// TIA Portal project "Proyecto Recreo OP 666" (V17)

(* hardware
DEVICE "S7-1200 station_1"  S7-1200 Station
   slot 0: "Rack_0"  S7-1200 Rack  Rack  V1.0
   slot 1: "PLC_1"  CPU 1214C DC/DC/DC  6ES7 214-1AG40-0XB0  V4.5
   slot 2: "DI 16/DQ 16x24VDC_1"  SM 1223 DI16/DQ16 x 24VDC  6ES7 223-1BL30-0XB0  V1.0
   slot 3: "AI 8x13BIT_1"  6ES7 231-4HF32-0XB0  V2.1
DEVICE "HMI_1"  KTP900 Basic PN
   slot 0: "HMI_1"  KTP900 Basic PN  6AV2 123-2JB03-0AX0  17.0.0.0
   slot 1: "HMI_RT_1"  KTP900 Basic PN  6AV2 123-2JB03-0AX0  17.0.0.0
   slot 5: "HMI_1.IE_CP_1"  PROFINET Interface  17.0.0.0
      slot 1: "PROFINET Interface_1"  PROFINET Interface
         slot 1: "Port_1"  Port
*)

// ===== PLC "PLC_1"  CPU 1214C DC/DC/DC =====

VAR_GLOBAL   // PLC tag table "BOOLEANAS"
   "HMI INICIAR CICLO PO" AT %M300.0 : Bool;
   "HMI INICIAR CICLO OP" AT %M300.3 : Bool;
   "HMI ON MANUAL VS" AT %M300.4 : Bool;
   "HMI ON MANUAL VV" AT %M300.5 : Bool;
   "HMI ON MANUAL CARGA AGUA" AT %M300.6 : Bool;
   "HMI ON MANUAL TOMA FILTRO" AT %M300.7 : Bool;
   "HMI ON MANUAL BALIZA VERDE" AT %M301.0 : Bool;
   "HMI ON MANUAL BALIZA ROJA" AT %M301.1 : Bool;
   "HMI ON MANUAL BUZZER" AT %M301.2 : Bool;
   "HMI SIGUIENTE EQUIPO MM" AT %M302.2 : Bool;   // Siguiente equipo modo manual
   "HMI ANTERIOR EQUIPO MM" AT %M302.3 : Bool;   // Anterior equipo modo manual
   "HMI OFF MANUAL VS" AT %M301.3 : Bool;
   "HMI OFF MANUAL VV" AT %M301.4 : Bool;
   "HMI OFF MANUAL CARGA AGUA" AT %M301.5 : Bool;
   "HMI OFF MANUAL TOMA FILTRO" AT %M301.6 : Bool;
   "HMI OFF MANUAL BALIZA VERDE" AT %M301.7 : Bool;
   "HMI OFF MANUAL BALIZA ROJA" AT %M302.0 : Bool;
   "HMI OFF MANUAL BUZZER" AT %M302.1 : Bool;
   "HMI ON MANUAL BOMBA RECIRCULACION" AT %M302.4 : Bool;
   "HMI OFF MANUAL BOMBA RECIRCULACION" AT %M302.5 : Bool;
   "HMI PAUSA" AT %M302.6 : Bool;
   "HMI CONTINUAR" AT %M302.7 : Bool;
   "HMI CANCELAR" AT %M303.0 : Bool;
   "HMI VER EQUIPO 1" AT %M303.1 : Bool;
   "HMI VER EQUIPO 2" AT %M303.2 : Bool;
   "HMI VER EQUIPO 3" AT %M303.3 : Bool;
   "HMI VER EQUIPO 4" AT %M303.4 : Bool;
   "ACTUALIZAR DATOS" AT %M303.5 : Bool;
   "HMI AUMENTAR CANT TORRES" AT %M303.6 : Bool;
   "HMI DISMINUIR CANT TORRES" AT %M303.7 : Bool;
   "HMI AUMENTAR EQUIPO" AT %M305.0 : Bool;
   "HMI DISMINUIR EQUIPO" AT %M305.1 : Bool;
   "HMI RECETA SIGUIENTE" AT %M305.2 : Bool;
   "HMI RECETA ANTERIOR" AT %M305.3 : Bool;
   "AUX 1" AT %M305.4 : Bool;
   "HMI SUMAR PASO" AT %M305.5 : Bool;
   "HMI RESTAR PASO" AT %M305.6 : Bool;
   "ACTUALIZAR RECETA" AT %M306.0 : Bool;
   "HMI SEL SIG RECETA" AT %M304.0 : Bool;
   "HMI SEL ANT RECETA" AT %M304.1 : Bool;
   "AUX 2" AT %M304.2 : Bool;
   "HMI ON BUZZER" AT %M304.3 : Bool;
   "HMI OFF BUZZER" AT %M304.4 : Bool;
   "CALIBRACION SN MAXIMO" AT %M304.5 : Bool;
   "CALIBRACION SN MINIMO" AT %M304.6 : Bool;
   "REARMADO" AT %M304.7 : Bool;
   "HMI ON LUZ PS REARME" AT %M305.7 : Bool;
   "HMI OFF LUZ PS REARME" AT %M306.1 : Bool;
   "Clock_Byte" AT %MB1500 : Byte;
   "Clock_10Hz" AT %M1500.0 : Bool;
   "Clock_5Hz" AT %M1500.1 : Bool;
   "Clock_2.5Hz" AT %M1500.2 : Bool;
   "Clock_2Hz" AT %M1500.3 : Bool;
   "Clock_1.25Hz" AT %M1500.4 : Bool;
   "Clock_1Hz" AT %M1500.5 : Bool;
   "Clock_0.625Hz" AT %M1500.6 : Bool;
   "Clock_0.5Hz" AT %M1500.7 : Bool;
   "HMI ON LUZ REARME" AT %M1501.0 : Bool;
   "HMI OFF LUZ REARME" AT %M1501.1 : Bool;
   "HMI ON INGRESO AMONIACO" AT %M306.2 : Bool;
   "HMI OFF INGRESO AMONIACO" AT %M306.3 : Bool;
   "HMI ON MANUAL V INGRESO" AT %M306.4 : Bool;
   "HMI OFF MANUAL V INGRESO" AT %M306.5 : Bool;
   "HMI ON MANUAL BI" AT %M306.6 : Bool;
   "HMI OFF MANUAL BI" AT %M306.7 : Bool;
   "HMI ON MANUAL BE" AT %M307.0 : Bool;
   "HMI OFF MANUAL BE" AT %M307.1 : Bool;
   "TIPO DE EQUIPO SELECCIONADO" AT %M307.2 : Bool;
   "HMI OK FIN DE CICLO" AT %M307.3 : Bool;
   "HMI OK CANCELAR" AT %M307.4 : Bool;
   "BLOQUEO" AT %M307.5 : Bool;
   "HMI RESET ACTUADORES MANUAL" AT %M307.6 : Bool;
   "HMI SALTAR PASO" AT %M307.7 : Bool;
   "BUZZER EQ1" AT %M308.0 : Bool;
   "BUZZER EQ2" AT %M308.1 : Bool;
   "BUZZER EQ3" AT %M308.2 : Bool;
   "BUZZER EQ4" AT %M308.3 : Bool;
   "System_Byte" AT %MB1700 : Byte;
   "FirstScan" AT %M1700.0 : Bool;
   "DiagStatusUpdate" AT %M1700.1 : Bool;
   "AlwaysTRUE" AT %M1700.2 : Bool;
   "AlwaysFALSE" AT %M1700.3 : Bool;
   "HMI VISUALIZAR RECETA" AT %M1701.0 : Bool;
   "HMI RECETARIO" AT %M1701.1 : Bool;
   "HMI VOLVER" AT %M1701.2 : Bool;
   "HMI ON LEVANTAR TAPA" AT %M1701.3 : Bool;
   "HMI OFF LEVANTAR TAPA" AT %M1701.4 : Bool;
   "HMI ON BAJAR TAPA" AT %M1701.5 : Bool;
   "HMI OFF BAJAR TAPA" AT %M1701.6 : Bool;
   "HMI CONFIRMAR LOTE" AT %M1701.7 : Bool;
END_VAR

VAR_GLOBAL   // PLC tag table "ENTERAS"
   "EQUIPO SELECCIONADO" AT %MW700 : Int;
   "EQUIPO ACTUAL" AT %MW702 : Int;
   "TORRES SELECCIONADAS" AT %MW704 : Int;
   "TORRES ACTUAL" AT %MW706 : Int;
   "CANT TORRES" AT %MW708 : Int;
   "EQUIPO MANUAL" AT %MW710 : Int;
   "AUXILIAR 1" AT %MW712 : Int;
   "AUXILIAR 2" AT %MW714 : Int;
   "AUXILIAR 3" AT %MW716 : Int;
   "AUXILIAR 4" AT %MW718 : Int;
   "AUXILIAR 5" AT %MW720 : Int;
   "TEMP CORTE PC" AT %MW726 : Int;
   "TIEMPO CORTE PC" AT %MW728 : Int;
   "CORTE PC POR TEMP" AT %MW730 : Int;
   "CORTE PC POR TIEMPO" AT %MW732 : Int;
   "DELAY" AT %MW734 : Int;
   "NM_CT" AT %MW736 : Int;   // Nivel minimo segun cantidad de torres
   "CTD PASADAS" AT %MW738 : Int;   // Cantidad de pasadas
   "FLAG CR" AT %MW740 : Int;   // Flag calculos realizados
   "HMI NUMERO RECETA" AT %MW742 : Int;
   "EQUIPO ACTUAL CALCULO" AT %MW744 : Int;
   "HMI RECETA SELECCIONADA" AT %MW746 : Int;
   "HMI NIVEL" AT %MW748 : Int;
   "AUXILIAR 6" AT %MW750 : Int;
   "VER NUMERO RECETA" AT %MW752 : Int;
   "VALOR CONTRASEÑA CALCULADA" AT %MD754 : DInt;
   "HMI CONTRASEÑA INGRESADA" AT %MD758 : DInt;
   "DIAS RESTANTES" AT %MD762 : DInt;
   "DIAS TRANSCURRIDOS" AT %MD766 : DInt;
   "IMAGEN BLOQUEO" AT %MW770 : Int;
   "AUX REC SEL" AT %MW772 : Int;
   "AUX NUM REC" AT %MW774 : Int;
END_VAR

VAR_GLOBAL   // PLC tag table "Entradas Analogicas"
   "PT100 agua EQ1" AT %IW96 : Int;
   "PT100 ingreso EQ1" AT %IW98 : Int;
   "PT100 producto EQ1" AT %IW100 : Int;
   "Regla nivel EQ1" AT %IW64 : Int;
   "PT100 agua EQ2" AT %IW104 : Int;
   "PT100 ingreso EQ2" AT %IW106 : Int;
   "PT100 producto EQ2" AT %IW108 : Int;
   "Regla nivel EQ2" AT %IW66 : Int;
END_VAR

VAR_GLOBAL   // PLC tag table "Salidas digitales"
   "C1 VS" AT %Q20.3 : Bool;
   "C1 VV" AT %Q20.4 : Bool;
   "C1 CARGA DE AGUA" AT %Q20.1 : Bool;
   "C1 BOMBA" AT %Q20.0 : Bool;
   "C1 BALIZA ROJA" AT %Q0.0 : Bool;
   "C1 BALIZA VERDE" AT %Q0.1 : Bool;
   "BUZZER" AT %Q0.4 : Bool;
   "C1 TOMA FILTRO" AT %Q20.2 : Bool;
   "LUZ PS REARME" AT %Q0.5 : Bool;
   "E1 BALIZA ROJA" AT %Q0.2 : Bool;
   "E1 BALIZA VERDE" AT %Q0.3 : Bool;
   "E1 CARGA DE AGUA" AT %Q20.6 : Bool;
   "E1 TOMA FILTRO" AT %Q20.7 : Bool;
   "E1 BOMBA" AT %Q20.5 : Bool;
   "E1 INGRESO AMONIACO" AT %Q21.0 : Bool;
   "LEVANTAR TAPA" AT %Q21.1 : Bool;   // VER DIRECCION
   "CERRAR TAPA" AT %Q0.6 : Bool;   // VER DIRECCION
END_VAR

VAR_GLOBAL   // PLC tag table "Entradas digitales"
   "VVC_C" AT %I0.2 : Bool;   // True en Reposo
   "VVA_C" AT %I0.3 : Bool;   // True cuando esta activada
   "VSC_C" AT %I0.6 : Bool;   // True en reposo
   "VSA_C" AT %I0.7 : Bool;   // True cuando esta activada
   "ESTADO REARME" AT %I6.0 : Bool;   // Estado de rearme ( Circuito si o no rearmado)
   "PRARM" AT %I1.0 : Bool;   // Pulsador de rearme
   "PEMERG" AT %I1.2 : Bool;   // Pulsador parada de emergencia
   "CH_F_E" AT %I1.3 : Bool;   // Falla chiller enfriador
   "GM_E" AT %I20.0 : Bool;   // Guardamotor bomba enfriador
   "GM_C" AT %I20.1 : Bool;   // Guardamotor bomba cocina
   "PS SUBIR TAPA" AT %I20.2 : Bool;
   "PS BAJAR TAPA" AT %I20.3 : Bool;
END_VAR

DATA_BLOCK "FUNCION EQUIPO_DB"   // DB2
{ S7_Optimized_Access := 'TRUE' }
VERSION : 0.1
// stored: InstanceOfName FUNCION EQUIPO
"FUNCION EQUIPO"
BEGIN
END_DATA_BLOCK

DATA_BLOCK "NOMBRE DE LOS EQUIPOS"   // DB3
{ S7_Optimized_Access := 'TRUE' }
VERSION : 0.1
   VAR
      EQUIPOS : Array[1..2] of String;
   END_VAR
BEGIN
   EQUIPOS[1] := 'COCINA 1';
   EQUIPOS[2] := 'ENFRIADOR 1';
END_DATA_BLOCK

DATA_BLOCK "ESTRUCTURAS Y ARREGLOS"   // DB4
{ S7_Optimized_Access := 'TRUE' }
VERSION : 0.1
   VAR
      TEMPERATURAS : Array[1..2] of Struct
         "TEMPERATURA AGUA" : Real;
         "TEMPERATURA INGRESO" : Real;
         "TEMPERATURA PRODUCTO" : Real;
         "TEMPERATURA AGUA SC" : Real;
         "TEMPERATURA INGRESO SC" : Real;
         "TEMPERATURA PRODUCTO SC" : Real;
      END_STRUCT;
      NIVEL : Array[1..2] of Int;
   END_VAR
   VAR RETAIN
      CORRECCIONES : Array[1..2] of Struct
         "TEMPERATURA AGUA" : Real;
         "TEMPERATURA INGRESO" : Real;
         "TEMPERATURA PRODUCTO" : Real;
      END_STRUCT;
   END_VAR
   VAR
      "NIVEL ALCANZADO" : Array[1..2] of Bool;
   END_VAR
   VAR RETAIN
      "TEMP CORTE PO" : Array[1..4] of Int;
      CONFIGURACION : Array[1..2] of Struct
         DELAY : Int;
         HISTERESIS : DInt;
         "TIEMPO MAXIMO CICLO" : Int;
         "NIVEL CRITICO PO" : Int;
         "NIVEL PO" : Array[1..3] of Int;
         "NIVEL OP" : Int;
         VENTANA : Int;
         "NIVEL CRITICO OP" : Int;
      END_STRUCT;
   END_VAR
   VAR
      "HMI CONFIGURACION" : Struct
         DELAY : Int;
         HISTERESIS : DInt;
         "TIEMPO MAXIMO CICLO" : Int;
         "NIVEL CRITICO PO" : Int;
         "NIVEL PO" : Array[1..3] of Int;
         "NIVEL OP" : Int;
         VENTANA : Int;
         "NIVEL CRITICO OP" : Int;
      END_STRUCT;
   END_VAR
   VAR RETAIN
      CARGA : Array[1..2] of Struct   // Lo traslado a cada equipo desde HMI carga
         "CANTIDAD DE TORRES" : Int;
         "NIVEL MINIMO" : Array[1..3] of Int;   // El arreglo es porque hay 3 torres
         "TIPO DE CORTE" : Bool;
         "TEMPERATURA CORTE PC" : Int;
         "TIEMPO CORTE PC" : Int;
         "NUMERO RECETA" : Int;
         "NOMBRE RECETA" : String;
         "ESTADO ACTUAL" : String;
         "TIEMPO TOTAL TRANSCURRIDO" : Int;
         "PASO ACTUAL" : Int;
         "VAPOR VIVO" : Bool;
      END_STRUCT;
   END_VAR
   VAR
      "HMI CARGA" : Struct   // Lo que veo en la pantalla cuando selecciono cada equipo (comun a todos)
         TEMPERATURAS : Struct
            "TEMPERATURA AGUA" : Real;
            "TEMPERATURA INGRESO" : Real;
            "TEMPERATURA PRODUCTO" : Real;
            "TEMPERATURA AGUA SC" : Real;
            "TEMPERATURA INGRESO SC" : Real;
            "TEMPERATURA PRODUCTO SC" : Real;
         END_STRUCT;
         NIVEL : Int;
         "CANTIDAD DE TORRES" : Int := 1;
         "NIVEL MINIMO" : Int;
         "TIPO DE CORTE" : Bool;
         "TEMPERATURA CORTE PC" : Int;
         "TIEMPO CORTE PC" : Int;
         "NUMERO RECETA" : Int;
         "NOMBRE RECETA" : String;
         "ESTADO ACTUAL" : String;
         "TIEMPO TOTAL TRANSCURRIDO" : Int;
         "PASO ACTUAL" : Int;
         "VAPOR VIVO" : Bool;
      END_STRUCT;
      "HMI EDICION RECETAS" : Struct
         PASOS : Int;
         "TEMP AGUA" : Array[1..4] of Int;
         "TEMP PRODUCTO" : Array[1..4] of Int;
         "TIEMPO CORTE" : Array[1..4] of Int;
         "TIPO CORTE" : Array[1..4] of Bool;
         NOMBRE : String;
         "TIEMPO CORTE ENFRIADO" : Int;
         "TEMP CORTE ENFRIADO" : Int;
         "TIPO CORTE ENFRIADO" : Bool;
      END_STRUCT;
   END_VAR
   VAR RETAIN
      RECETARIO : Array[0..20] of Struct
         PASOS : Int;
         "TEMP AGUA" : Array[1..4] of Int;
         "TEMP PRODUCTO" : Array[1..4] of Int;
         "TIEMPO CORTE" : Array[1..4] of Int;
         "TIPO CORTE" : Array[1..4] of Bool;
         NOMBRE : String;
         "TIEMPO CORTE ENFRIADO" : Int;
         "TEMP CORTE ENFRIADO" : Int;
         "TIPO CORTE ENFRIADO" : Bool;
      END_STRUCT;
      "CARGA RECETA" : Array[1..2] of Struct   // Se guarda la receta elegida en cada equipo
         PASOS : Int;
         "TEMP AGUA" : Array[1..4] of Int;
         "TEMP PRODUCTO" : Array[1..4] of Int;
         "TIEMPO CORTE" : Array[1..4] of Int;
         "TIPO CORTE" : Array[1..4] of Bool;
         NOMBRE : String;
         "TIEMPO CORTE ENFRIADO" : Int;
         "TEMP CORTE ENFRIADO" : Int;
         "TIPO CORTE ENFRIADO" : Bool;
      END_STRUCT;
      "CARGA NUMERO RECETA" : Array[0..4] of Int;   // *********** CUIDADOOOO
   END_VAR
   VAR
      "CORRECCIONES HMI" : Struct
         "TEMPERATURA AGUA SC" : Real;
         "TEMPERATURA INGRESO SC" : Real;
         "TEMPERATURA PRODUCTO SC" : Real;
      END_STRUCT;
      "CALIBRAR MINIMO SN" : Array[1..2] of Bool;
      "CALIBRAR MAXIMO SN" : Array[1..2] of Bool;
      "HMI MOSTRAR RECETA" : Struct
         PASOS : Int;
         "TEMP AGUA" : Array[1..4] of Int;
         "TEMP PRODUCTO" : Array[1..4] of Int;
         "TIEMPO CORTE" : Array[1..4] of Int;
         "TIPO CORTE" : Array[1..4] of Bool;
         NOMBRE : String;
         "TIEMPO CORTE ENFRIADO" : Int;
         "TEMP CORTE ENFRIADO" : Int;
         "TIPO CORTE ENFRIADO" : Int;
      END_STRUCT;
      "HMI ESTADO" : Struct
         EQUIPO : String;
         CHILLER : String;
         "COLOR EN HMI" : Int;
         "TIEMPO TRANSCURRIDO" : DInt;
         "EN PO" : Bool;
         "EN OP" : Bool;
         "EN CICLO" : Bool;
         "TIPO DE CORTE" : String;
         "PULSADOR PAUSA" : Bool;
         "PULSADOR CONTINUAR" : Bool;
         "PULSADOR CANCELAR" : Bool;
         "CICLO CANCELADO" : Bool;
         "CICLO FINALIZADO" : Bool;
         "PULSADOR CICLO CANCELADO" : Bool;
         "PULSADOR CICLO FINALIZADO" : Bool;
         "RESET ACTUADORES" : Bool;
         "MANUAL ACTIVO" : Bool;
         "PASO ACTUAL" : Int;
      END_STRUCT;
      ESTADO : Array[1..2] of Struct
         EQUIPO : String;
         CHILLER : String;
         "COLOR EN HMI" : Int;
         "TIEMPO TRANSCURRIDO" : DInt;
         "EN PO" : Bool;
         "EN OP" : Bool;
         "EN CICLO" : Bool;
         "TIPO DE CORTE" : String;
         "PULSADOR PAUSA" : Bool;
         "PULSADOR CONTINUAR" : Bool;
         "PULSADOR CANCELAR" : Bool;
         "CICLO CANCELADO" : Bool;
         "CICLO FINALIZADO" : Bool;
         "PULSADOR CICLO CANCELADO" : Bool;
         "PULSADOR CICLO FINALIZADO" : Bool;
         "RESET ACTUADORES" : Bool;
         "MANUAL ACTIVO" : Bool;
         "PASO ACTUAL" : Int;
         "CONFIRMACION LOTE" : Bool;
      END_STRUCT;
      "HMI NOMBRE EQUIPO" : String;
   END_VAR
BEGIN
   CARGA[1]."CANTIDAD DE TORRES" := 1;
   CARGA[2]."CANTIDAD DE TORRES" := 1;
   CONFIGURACION[1]."NIVEL PO"[1] := 1020;   // Nivel PO para 1 torre
   CONFIGURACION[1]."NIVEL PO"[2] := 825;   // Nivel PO para 2 torres
   CONFIGURACION[1]."NIVEL PO"[3] := 700;   // Nivel PO para 3 torres
   CONFIGURACION[1].HISTERESIS := 2;
   CONFIGURACION[1]."TIEMPO MAXIMO CICLO" := 400;
   CONFIGURACION[2].HISTERESIS := 2;
   CONFIGURACION[2]."TIEMPO MAXIMO CICLO" := 400;
   CONFIGURACION[2]."NIVEL PO"[1] := 1020;
   CONFIGURACION[2]."NIVEL PO"[2] := 825;
   CONFIGURACION[2]."NIVEL PO"[3] := 700;
   CONFIGURACION[1]."NIVEL OP" := 1163;
   CONFIGURACION[2]."NIVEL OP" := 1163;
   CONFIGURACION[2]."NIVEL CRITICO PO" := 550;
   CONFIGURACION[2]."NIVEL CRITICO OP" := 985;
   // "HMI CONFIGURACION"."NIVEL PO"[1] : Nivel para 1 torre
   // "HMI CONFIGURACION"."NIVEL PO"[2] : Nivel para 2 torres
   // "HMI CONFIGURACION"."NIVEL PO"[3] : Nivel para 3 torres
   // CARGA[1] : Cada equipo con sus configuraciones en
END_DATA_BLOCK

DATA_BLOCK "ALARMAS"   // DB5
{ S7_Optimized_Access := 'FALSE' }
VERSION : 0.1
   VAR
      COCINAS : Struct
         "FALLA VALVULA VAPOR SERPENTINA" : Bool;
         "FALLA VALVULA VAPOR VIVO" : Bool;
         "FALLA GUARDAMOTOR" : Bool;
         "NIVEL CRITICO" : Bool;
         "FALLA SENSOR TEMP AGUA" : Bool;
         "FALLA SENSOR TEMP INGRESO" : Bool;
         "FALLA SENSOR TEMP PRODUCTO" : Bool;
         "TIEMPO MAXIMO CARGA DE AGUA" : Bool;
      END_STRUCT;
      ENFRIADOR : Struct
         "FALLA GUARDAMOTOR" : Bool;
         "FALLA CHILLER" : Bool;
         "NIVEL CRITICO" : Bool;
         "FALLA SENSOR TEMP AGUA" : Bool;
         "FALLA SENSOR TEMP INGRESO" : Bool;
         "FALLA SENSOR TEMP PRODUCTO" : Bool;
         "TIEMPO MAXIMO CARGA DE AGUA" : Bool;
      END_STRUCT;
      "PULSADOR EM ACTIVO" : Bool;
      "PRESIONAR PULSADOR REARME" : Bool;
   END_VAR
BEGIN
END_DATA_BLOCK

DATA_BLOCK "ENTRADAS Y SALIDAS"   // DB6
{ S7_Optimized_Access := 'TRUE' }
VERSION : 0.1
   VAR
      "VV MANUAL" : Array[1..2] of Bool;
      "VS MANUAL" : Array[1..2] of Bool;
      "CARGA AGUA MANUAL" : Array[1..2] of Bool;
      "TOMA FILTRO MANUAL" : Array[1..2] of Bool;
      "BOMBA RECIRCULACION MANUAL" : Array[1..2] of Bool;
      "BALIZA VERDE MANUAL" : Array[1..2] of Bool;
      "BALIZA ROJA MANUAL" : Array[1..2] of Bool;
      "INGRESO AMONIACO MANUAL" : Array[1..2] of Bool;
      "LEVANTAR TAPA MANUAL" : Array[1..2] of Bool;
      "BAJAR TAPA MANUAL" : Array[1..2] of Bool;
      "INGRESO AMONIACO" : Array[1..2] of Bool;
      GUARDAMOTOR : Array[1..2] of Bool;
      "SERPENTINA ABIERTA" : Array[1..2] of Bool;
      "SERPENTINA CERRADA" : Array[1..2] of Bool;
      "VAPOR VIVO ABIERTO" : Array[1..2] of Bool;
      "VAPOR VIVO CERRADO" : Array[1..2] of Bool;
      "FALLA CHILLER" : Array[1..2] of Bool;
      "BUZZER MANUAL" : Bool;
      "LUZ MANUAL PS REARME" : Bool;
   END_VAR
BEGIN
END_DATA_BLOCK

DATA_BLOCK "ESTADO"   // DB7
{ S7_Optimized_Access := 'TRUE' }
VERSION : 0.1
   VAR
      SALIDAS : Struct
         COCINAS : Array[1..2] of Struct
            "BALIZA VERDE" : Bool;
            "BALIZA ROJA" : Bool;
            "BOMBA RECIRCULACION" : Bool;
            "CARGA DE GUA" : Bool;
            "TOMA FILTRO" : Bool;
            "VAPOR SERPENTINA" : Bool;
            "VAPOR VIVO" : Bool;
         END_STRUCT;
         ENFRIADORES : Array[1..2] of Struct
            "BALIZA VERDE" : Bool;
            "BALIZA ROJA" : Bool;
            "BOMBA RECIRCULACION" : Bool;
            "CARGA DE AGUA" : Bool;
            "TOMA FILTRO" : Bool;
            "INGRESO AMONIACO" : Bool;
         END_STRUCT;
      END_STRUCT;
      ENTRADAS : Struct
         COCINAS : Array[1..2] of Struct
            GUARDAMOTOR : Bool;
            "VAPOR VIVO CERRADO" : Bool;
            "VAPOR VIVO ABIERTO" : Bool;
            "SERPENTINA CERRADA" : Bool;
            "SERPENTINA ABIERTA" : Bool;
         END_STRUCT;
         ENFRIADORES : Array[1..2] of Struct
            GUARDAMOTOR : Bool;
            "FALLA CHILLER" : Bool;
         END_STRUCT;
      END_STRUCT;
   END_VAR
BEGIN
END_DATA_BLOCK

DATA_BLOCK "VISUALIZACIONES HMI"   // DB8
{ S7_Optimized_Access := 'TRUE' }
VERSION : 0.1
   VAR
      "ON VS" : Bool;
      "OFF VS" : Bool;
      "ON VV" : Bool;
      "OFF VV" : Bool;
      "ON/OFF CARGA AGUA" : Bool;
      "ON/OFF TOMA FILTRO" : Bool;
      "ON/OFF BOMBA RECIRCULACION" : Bool;
      "ON/OFF BV" : Bool;
      "ON/OFF BR" : Bool;
      "ON BOMBA INGRESO" : Bool;
      "OFF BOMBA INGRESO" : Bool;
      "ON BOMBA EGRESO" : Bool;
      "OFF BOMBA EGRESO" : Bool;
      "ON V INGRESO" : Bool;
      "OFF V INGRESO" : Bool;
      "ON V EGRESO" : Bool;
      "OFF V EGRESO" : Bool;
      "ON SUBIR TAPA" : Bool;
      "OFF SUBIR TAPA" : Bool;
      "ON BAJAR TAPA" : Bool;
      "OFF BAJAR TAPA" : Bool;
      "ON INGRESO AMONIACO" : Bool;
      "OFF INGRESO AMONIACO" : Bool;
      BUZZER : Bool;
      "GUARDAMOTOR BOMBA REC" : Bool;
      "SERPENTINA CERRADA" : Bool;
      "SERPENTINA ABIERTA" : Bool;
      "VAPOR VIVO CERRADO" : Bool;
      "VAPOR VIVO ABIERTO" : Bool;
      "NV CHILLER REBALSE" : Bool;
      "NV CHILLER OK" : Bool;
      "NV CHILLER BAJO" : Bool;
      "GUARDAMOTOR BOMBA INGRESO" : Bool;
      "GUARDAMOTOR BOMBA EGRESO" : Bool;
      "FALLA CHILLER" : Bool;
      "1 PASO RECETA" : Bool;
      "2 PASOS RECETA" : Bool;
      "3 PASOS RECETA" : Bool;
      "4 PASOS RECETA" : Bool;
      "CORTE TEMP PASO 1" : Bool;
      "CORTE TEMP PASO 2" : Bool;
      "CORTE TEMP PASO 3" : Bool;
      "CORTE TEMP PASO 4" : Bool;
      "CORTE TIEMPO PASO 1" : Bool;
      "CORTE TIEMPO PASO 2" : Bool;
      "CORTE TIEMPO PASO 3" : Bool;
      "CORTE TIEMPO PASO 4" : Bool;
      "CORTE TEMP ENFRIADOR" : Bool;
      "CORTE TIEMPO ENFRIADOR" : Bool;
      "PASOS OP EN COCINAS" : Bool;
      GRAFICOS : Int;
      "LIM SUP CANT TORRES" : Bool;
      "LIM INF CANT TORRES" : Bool;
      "LIM SUP EQUIPO SEL" : Bool;
      "LIM INF EQUIPO SEL" : Bool;
      "EN VISUALIZAR RECETA" : Bool;
      "EN RECETARIO" : Bool;
      "SIGUIENTE RECETA" : Bool;
      "ANTERIOR RECETA" : Bool;
      "SIGUIENTE PASO" : Bool;
      "ANTERIOR PASO" : Bool;
      "BLOQUEO EDICION RECETAS" : Bool;
   END_VAR
BEGIN
END_DATA_BLOCK

DATA_BLOCK "SELECCION DE EQUIPO_DB"   // DB9
{ S7_Optimized_Access := 'TRUE' }
VERSION : 0.1
// stored: InstanceOfName SELECCION DE EQUIPO
"SELECCION DE EQUIPO"
BEGIN
END_DATA_BLOCK

DATA_BLOCK "EQUIPO 1"   // DB10
{ S7_Optimized_Access := 'TRUE' }
VERSION : 0.1
// stored: InstanceOfName NIVEL DE AGUA
"NIVEL DE AGUA"
BEGIN
END_DATA_BLOCK

DATA_BLOCK "EQUIPO 2"   // DB14
{ S7_Optimized_Access := 'TRUE' }
VERSION : 0.1
// stored: InstanceOfName NIVEL DE AGUA
"NIVEL DE AGUA"
BEGIN
END_DATA_BLOCK

DATA_BLOCK "EQUIPO 3"   // DB15
{ S7_Optimized_Access := 'TRUE' }
VERSION : 0.1
// stored: InstanceOfName NIVEL DE AGUA
"NIVEL DE AGUA"
BEGIN
END_DATA_BLOCK

DATA_BLOCK "EQUIPO 4"   // DB16
{ S7_Optimized_Access := 'TRUE' }
VERSION : 0.1
// stored: InstanceOfName NIVEL DE AGUA
"NIVEL DE AGUA"
BEGIN
END_DATA_BLOCK

DATA_BLOCK "EQUIPO_3"   // DB17
{ S7_Optimized_Access := 'TRUE' }
VERSION : 0.1
// stored: InstanceOfName ENFRIADOR
"ENFRIADOR"
BEGIN
END_DATA_BLOCK

DATA_BLOCK "SENSADO ENTRADA FUNCION"   // DB18
{ S7_Optimized_Access := 'TRUE' }
VERSION : 0.1
   VAR
      ENFRIADORES : Struct
         "GUARDAMOTOR BI" : Array[1..4] of Bool;
         "GUARDAMOTOR BE" : Array[1..4] of Bool;
         "NIVEL BAJO CHILLER" : Array[1..4] of Bool;
         "NIVEL OK CHILLER" : Array[1..4] of Bool;
         "NIVEL REBALSE CHILLER" : Array[1..4] of Bool;
         "FALLA CHILLER" : Array[1..4] of Bool;
      END_STRUCT;
   END_VAR
BEGIN
END_DATA_BLOCK

DATA_BLOCK "EQUIPO_4"   // DB19
{ S7_Optimized_Access := 'TRUE' }
VERSION : 0.1
// stored: InstanceOfName ENFRIADOR
"ENFRIADOR"
BEGIN
END_DATA_BLOCK

DATA_BLOCK "EQUIPO_1"   // DB20
{ S7_Optimized_Access := 'TRUE' }
VERSION : 0.1
// stored: InstanceOfName COCINA
"COCINA"
BEGIN
END_DATA_BLOCK

DATA_BLOCK "EQUIPO_2"   // DB21
{ S7_Optimized_Access := 'TRUE' }
VERSION : 0.1
// stored: InstanceOfName COCINA
"COCINA"
BEGIN
END_DATA_BLOCK

DATA_BLOCK "Coordinacion"   // DB22
{ S7_Optimized_Access := 'TRUE' }
VERSION : 0.1
   VAR
      Comunicacion : Int;
   END_VAR
BEGIN
END_DATA_BLOCK

DATA_BLOCK "COMUNICACION"   // DB23
{ S7_Optimized_Access := 'TRUE' }
VERSION : 0.1
   VAR
      ESTADO : Int;
      "T AGUA" : Real;
      "T INGRESO" : Real;
      "T PROD" : Real;
      NIVEL : Int;
      "NOMBRE RECETA" : String;
      "NUMERO RECETA" : Int;
      "NUMERO EQUIPO" : Int;
      SERPENTINA : Bool;
      "VAPOR VIVO" : Bool;
      TORRES : Int;
      PASOS : Int;
      "TIEMPO TRANSCURRIDO" : DInt;
   END_VAR
BEGIN
END_DATA_BLOCK

DATA_BLOCK "ENVIO EQUIPO 1"   // DB24
{ S7_Optimized_Access := 'TRUE' }
VERSION : 0.1
// stored: InstanceOfName ENVIO DATOS
"ENVIO DATOS"
BEGIN
END_DATA_BLOCK

// folder: System blocks/Program resources

DATA_BLOCK "CANTIDAD TORRES"   // DB1
{ S7_Optimized_Access := 'TRUE' }
AUTHOR : Simatic
FAMILY : IEC
NAME : CNTR
VERSION : 1.0
// stored: InstanceOfName IEC_COUNTER
"IEC_COUNTER"
BEGIN
END_DATA_BLOCK

DATA_BLOCK "CONTADOR RECETAS"   // DB11
{ S7_Optimized_Access := 'TRUE' }
AUTHOR : Simatic
FAMILY : IEC
NAME : CNTR
VERSION : 1.0
// stored: InstanceOfName IEC_COUNTER
"IEC_COUNTER"
BEGIN
END_DATA_BLOCK

DATA_BLOCK "CONTADOR PASOS"   // DB12
{ S7_Optimized_Access := 'TRUE' }
AUTHOR : Simatic
FAMILY : IEC
NAME : CNTR
VERSION : 1.0
// stored: InstanceOfName IEC_COUNTER
"IEC_COUNTER"
BEGIN
END_DATA_BLOCK

DATA_BLOCK "CONTADOR SELECCION DE RECETA"   // DB13
{ S7_Optimized_Access := 'TRUE' }
AUTHOR : Simatic
FAMILY : IEC
NAME : CNTR
VERSION : 1.0
// stored: InstanceOfName IEC_COUNTER
"IEC_COUNTER"
BEGIN
END_DATA_BLOCK

// folder: (top level)

FUNCTION_BLOCK "ENFRIADOR"   // FB1, LAD
{ S7_Optimized_Access := 'TRUE' }
VERSION : 0.1
   VAR_INPUT
      REARME : Bool;
      "PARAMETROS CICLOS" : Struct
         "CANTIDAD DE TORRES" : Int;
         "NIVEL MINIMO" : Array[1..3] of Int;   // El arreglo es porque hay 3 torres
         "TIPO DE CORTE" : Bool;
         "TEMPERATURA CORTE PO" : Int;
         "TIEMPO CORTE PO" : Int;
         "NUMERO RECETA" : Int;
         "NOMBRE RECETA" : String;
         "ESTADO ACTUAL" : String;
         "TIEMPO TOTAL TRANSCURRIDO" : Int;
         "PASO ACTUAL" : Int;
         "VAPOR VIVO" : Bool;
      END_STRUCT;
      CONFIGURACION : Struct
         DELAY : Int;
         HISTERESIS : DInt;
         "TIEMPO MAXIMO CICLO" : Int;
         "NIVEL CRITICO" : Int;
         "NIVEL PO" : Array[1..3] of Int;
         "NIVEL OP" : Int;
         VENTANA : Int;
         "NIVEL CRITICO OP" : Int;
      END_STRUCT;
      RECETA : Struct
         PASOS : Int;
         "TEMP AGUA" : Array[1..4] of Int;
         "TEMP PRODUCTO" : Array[1..4] of Int;
         "TIEMPO CORTE" : Array[1..4] of Int;
         "TIPO CORTE" : Array[1..4] of Bool;
         NOMBRE : String;
         "TIEMPO CORTE ENFRIADO" : Int;
         "TEMP CORTE ENFRIADO" : Int;
         "TIPO CORTE ENFRIADO" : Bool;
      END_STRUCT;
      TEMPERATURAS : Struct
         "TEMPERATURA AGUA" : Real;
         "TEMPERATURA INGRESO" : Real;
         "TEMPERATURA PRODUCTO" : Real;
         "TEMPERATURA AGUA SC" : Real;
         "TEMPERATURA INGRESO SC" : Real;
         "TEMPERATURA PRODUCTO SC" : Real;
      END_STRUCT;
      NIVEL : Int;
      GUARDAMOTOR : Bool;
      "MANUAL BALIZA VERDE" : Bool;
      "MANUAL BALIZA ROJA" : Bool;
      "MANUAL BOMBA" : Bool;
      "MANUAL CARGA DE AGUA" : Bool;
      "MANUAL TOMA FILTRO" : Bool;
      "MANUAL INGRESO AMONIACO" : Bool;
      "EQUIPO SELECCIONADO" : Int;
      "NUMERO DE EQUIPO" : Int;
      "INICIAR PRE OPERATIVO" : Bool;
      "INICIAR OPERATIVO" : Bool;
      PAUSA : Bool;
      CONTINUAR : Bool;
      CANCELAR : Bool;
      "PULSADOR EMERGENCIA" : Bool;
      "OK FIN CICLO" : Bool;
      "OK CANCELAR" : Bool;
      "RESET ACTUADORES EN MANUAL" : Bool;
   END_VAR
   VAR_OUTPUT
      "BALIZA VERDE" : Bool;
      "BALIZA ROJA" : Bool;
      BUZER : Bool;
      BOMBA : Bool;
      "CARGA DE AGUA" : Bool;
      "TOMA FILTRO" : Bool;
      "INGRESO AMONIACO" : Bool;
      ESTADO : Struct
         EQUIPO : String;
         CHILLER : String;
         "COLOR EN HMI" : Int;
         "TIEMPO TRANSCURRIDO" : DInt;
         "EN PO" : Bool;
         "EN OP" : Bool;
         "EN CICLO" : Bool;
         "TIPO DE CORTE" : String;
         "PULSADOR PAUSA" : Bool;
         "PULSADOR CONTINUAR" : Bool;
         "PULSADOR CANCELAR" : Bool;
         "CICLO CANCELADO" : Bool;
         "CICLO FINALIZADO" : Bool;
         "PULSADOR CICLO CANCELADO" : Bool;
         "PULSADOR CICLO FINALIZADO" : Bool;
         "RESET ACTUADORES" : Bool;
         "MANUAL ACTIVO" : Bool;
         "PASO ACTUAL" : Int;
      END_STRUCT;
      ALARMAS : Struct
         "FALLA GUARDAMOTOR" : Bool;
         "FALLA CHILLER" : Bool;
         "NIVEL CRITICO TANQUE" : Bool;
         "FALLA SENSOR TEMP AGUA" : Bool;
         "FALLA SENSOR TEMP INGRESO" : Bool;
         "FALLA SENSOR TEMP PRODUCTO" : Bool;
         "TIEMPO MAXIMO CARGA DE AGUA" : Bool;
      END_STRUCT;
      "ESTADO ENTRADAS" : Struct
         GUARDAMOTOR : Bool;
         "FALLA CHILLER" : Bool;
      END_STRUCT;
      "ESTADO SALIDAS" : Struct
         "BALIZA VERDE" : Bool;
         "BALIZA ROJA" : Bool;
         "BOMBA RECIRCULACION" : Bool;
         "CARGA DE AGUA" : Bool;
         "TOMA FILTRO" : Bool;
         "INGRESO AMONIACO" : Bool;
      END_STRUCT;
   END_VAR
   VAR
      HABILITADO : Bool;
      "EN FALLA" : Bool;
      "CICLO PO ACTIVO" : Bool;
      "CICLO CANCELADO" : Bool;
      "CICLO PAUSADO" : Bool;
      "NIVEL PO" : Int;
      "TEMPERATURA PO ALCANZADA" : Bool;
      "TIEMPO PO" : TON_TIME;
      "TIEMPO CORTE PO" : DInt;
      "TIEMPO PO ALCANZADO" : Bool;
      "FIN CICLO PO" : Bool;
      "CICLO OP ACTIVO" : Bool;
      "TEMPERATURA OP ALCANZADA" : Bool;
      "TIEMPO OP" : TONR_TIME;
      "TIEMPO CORTE OP" : DInt;
      "FALTA AGUA PARA CHILLER" : Bool;
      "NIVEL CH CORRECTO COMIENZO" : Bool;
      "V EGRESO PARA CARGA CH" : Bool;
      "MANDAR AGUA A CH" : Bool;
      "CARGAR AGUA TQ PARA CARGA CH" : Bool;
      "CARGA AGUA TQ" : Bool;
      "NIVEL TQ ALCANZADO" : Bool;
      "NIVEL MINIMO" : Int;
      "NIVEL MAXIMO" : Int;
      "EN RANGO" : Bool;
      "NIVEL DEBAJO MINIMO" : Bool;
      "NIVEL SUPERA MAXIMO" : Bool;
      BOMBA_EGRESO : TON_TIME;
      BOMBA_INGRESO : TON_TIME;
      IEC_Timer_0_Instance : TOF_TIME;
      IEC_Timer_0_Instance_1 : TOF_TIME;
      DELAYS : DInt;
      "EN NIVEL PARA BI" : Bool;
      "EN NIVEL PARA BE" : Bool;
      "NIVEL TRABAJO" : Int;
      "NIVEL PARA CARGA DE AGUA" : Int;
      "TIEMPO OP ALCANZADO" : Bool;
      "FIN CICLO OP" : Bool;
      F1 : Bool;
      F2 : Bool;
      "TIEMPO MAXIMO" : DInt;
      AUXILIAR : DInt;
      IEC_Timer_0_Instance_2 : TONR_TIME;
      "CICLO PO FINALIZADO" : Bool;
      "CICLO OP FINALIZADO" : Bool;
      "ACTUADORES MANUALES ACTIVOS" : Bool;
      IEC_Timer_0_Instance_3 : TON_TIME;
      "FALLA SENSOR TEMPERATURA" : Bool;
      IEC_Timer_0_Instance_4 : TONR_TIME;
      "TIEMPO MAXIMO CARGA DE AGUA" : Bool;
      "NIVEL CRITICO PO" : Bool;
      "NIVEL CRITICO OP" : Bool;
      "CONTINUAR CICLO" : Bool;
      IEC_Timer_0_Instance_5 : TOF_TIME;
      F5 : Bool;
      F6 : Bool;
      F7 : Bool;
      F8 : Bool;
      IEC_Timer_0_Instance_6 : TOF_TIME;
      F9 : Bool;
      "TEMP MAXIMA" : Int;
      "TEMP MINIMA" : Int;
      "TEMP BAJA" : Bool;
      "TEMP EN RANGO" : Bool;
   END_VAR
   VAR CONSTANT
      "NIVEL MIN TQ PARA CARGA CH" : Int := 400;
      REBALSE : String := 'REBALSE';
      OK : String := 'OK';
      BAJO : String := 'BAJO';
      "PRE OPERACIONAL" : String := 'PRE OPERACIONAL';
      OPERACIONAL : String := 'OPERACIONAL';
      PAUSADO : String := 'PAUSADO';
      INACTIVO : String := 'INACTIVO';
      TEMPERATURA : String := 'TEMPERATURA';
      TIEMPO : String := 'TIEMPO';
      "NIVEL TOMA FILTRO" : Int := 550;
      "NIVEL FILTRO" : Int := 985;
   END_VAR
   VAR_TEMP   // added for the SCL form of the ladder/FBD networks
      _w1 : Bool;
      _w2 : Bool;
      _w3 : Bool;
      _w4 : Bool;
      _w5 : Bool;
   END_VAR
   // // CONFIGURACION."NIVEL PO"[1] : Nivel PO para 1 torre
   // // CONFIGURACION."NIVEL PO"[2] : Nivel PO para 2 torres
   // // CONFIGURACION."NIVEL PO"[3] : Nivel PO para 3 torres
BEGIN

REGION Network 1: HABILITACION
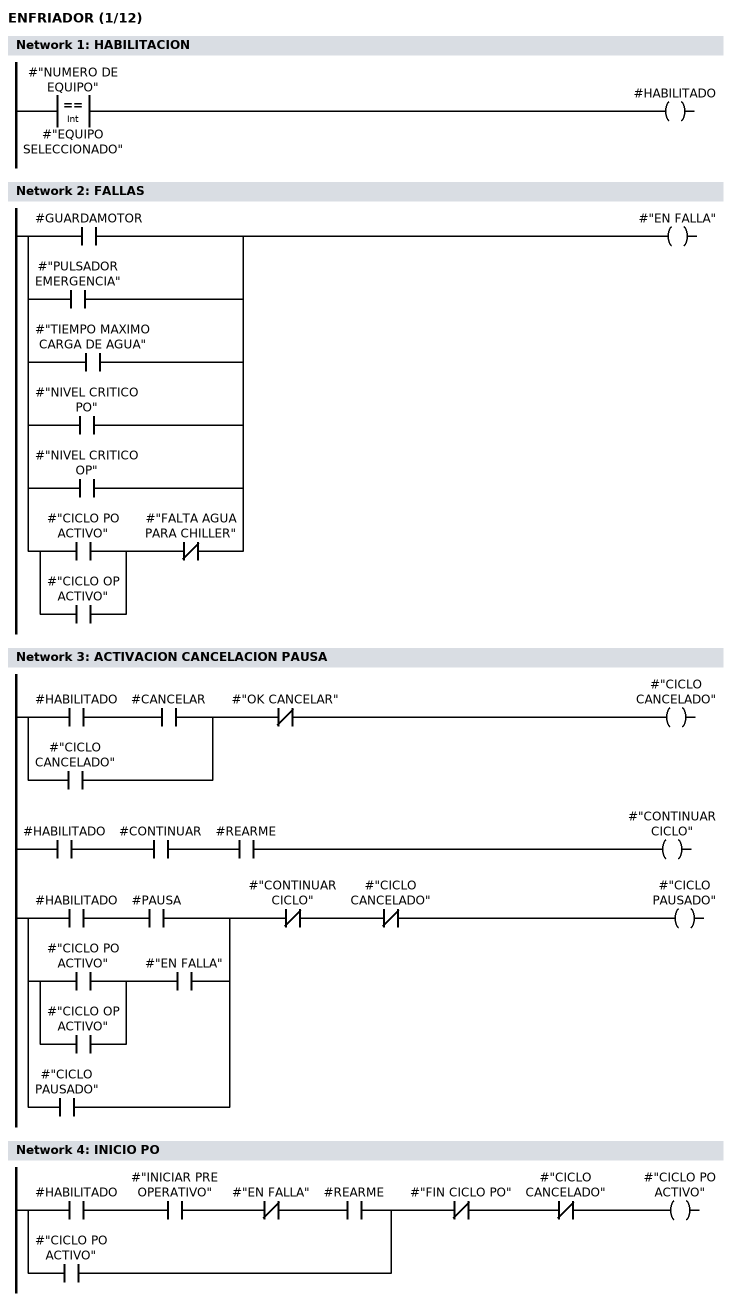
   RUNG wire#powerrail
      { S7_Templates := "SrcType := Int" } EQ_Contact(in1 := #"NUMERO DE EQUIPO", in2 := #"EQUIPO SELECCIONADO")
      Coil( #HABILITADO )
   END_RUNG
   // the same network as SCL:
   #HABILITADO := #"NUMERO DE EQUIPO" = #"EQUIPO SELECCIONADO";
END_REGION

REGION Network 2: FALLAS
   RUNG wire#powerrail
      Contact( #GUARDAMOTOR )
      wire#w1
      Coil( #"EN FALLA" )
   END_RUNG
   RUNG wire#powerrail
      Contact( #"PULSADOR EMERGENCIA" )
   END_RUNG wire#w1
   RUNG wire#powerrail
      Contact( #"TIEMPO MAXIMO CARGA DE AGUA" )
   END_RUNG wire#w1
   RUNG wire#powerrail
      Contact( #"NIVEL CRITICO PO" )
   END_RUNG wire#w1
   RUNG wire#powerrail
      Contact( #"NIVEL CRITICO OP" )
   END_RUNG wire#w1
   RUNG wire#powerrail
      Contact( #"CICLO PO ACTIVO" )
      wire#w2
      I_Contact( #"FALTA AGUA PARA CHILLER" )
   END_RUNG wire#w1
   RUNG wire#powerrail
      Contact( #"CICLO OP ACTIVO" )
   END_RUNG wire#w2
   // the same network as SCL:
   #"EN FALLA" := #GUARDAMOTOR OR #"PULSADOR EMERGENCIA" OR #"TIEMPO MAXIMO CARGA DE AGUA" OR #"NIVEL CRITICO PO" OR #"NIVEL CRITICO OP" OR ((#"CICLO PO ACTIVO" OR #"CICLO OP ACTIVO") AND NOT #"FALTA AGUA PARA CHILLER");
END_REGION

REGION Network 3: ACTIVACION CANCELACION PAUSA
   RUNG wire#powerrail
      Contact( #HABILITADO )
      Contact( #CANCELAR )
      wire#w1
      I_Contact( #"OK CANCELAR" )
      Coil( #"CICLO CANCELADO" )
   END_RUNG
   RUNG wire#powerrail
      Contact( #"CICLO CANCELADO" )
   END_RUNG wire#w1
   RUNG wire#powerrail
      Contact( #HABILITADO )
      Contact( #CONTINUAR )
      Contact( #REARME )
      Coil( #"CONTINUAR CICLO" )
   END_RUNG
   RUNG wire#powerrail
      Contact( #HABILITADO )
      Contact( #PAUSA )
      wire#w2
      I_Contact( #"CONTINUAR CICLO" )
      I_Contact( #"CICLO CANCELADO" )
      Coil( #"CICLO PAUSADO" )
   END_RUNG
   RUNG wire#powerrail
      Contact( #"CICLO PO ACTIVO" )
      wire#w3
      Contact( #"EN FALLA" )
   END_RUNG wire#w2
   RUNG wire#powerrail
      Contact( #"CICLO OP ACTIVO" )
   END_RUNG wire#w3
   RUNG wire#powerrail
      Contact( #"CICLO PAUSADO" )
   END_RUNG wire#w2
   // the same network as SCL:
   #"CICLO CANCELADO" := ((#HABILITADO AND #CANCELAR) OR #"CICLO CANCELADO") AND NOT #"OK CANCELAR";
   #"CONTINUAR CICLO" := #HABILITADO AND #CONTINUAR AND #REARME;
   #"CICLO PAUSADO" := ((#HABILITADO AND #PAUSA) OR ((#"CICLO PO ACTIVO" OR #"CICLO OP ACTIVO") AND #"EN FALLA") OR #"CICLO PAUSADO") AND NOT #"CONTINUAR CICLO" AND NOT #"CICLO CANCELADO";
END_REGION

REGION Network 4: INICIO PO
   RUNG wire#powerrail
      Contact( #HABILITADO )
      Contact( #"INICIAR PRE OPERATIVO" )
      I_Contact( #"EN FALLA" )
      Contact( #REARME )
      wire#w1
      I_Contact( #"FIN CICLO PO" )
      I_Contact( #"CICLO CANCELADO" )
      Coil( #"CICLO PO ACTIVO" )
   END_RUNG
   RUNG wire#powerrail
      Contact( #"CICLO PO ACTIVO" )
   END_RUNG wire#w1
   // the same network as SCL:
   #"CICLO PO ACTIVO" := ((#HABILITADO AND #"INICIAR PRE OPERATIVO" AND NOT #"EN FALLA" AND #REARME) OR #"CICLO PO ACTIVO") AND NOT #"FIN CICLO PO" AND NOT #"CICLO CANCELADO";
END_REGION

REGION Network 5: TOMA FILTRO
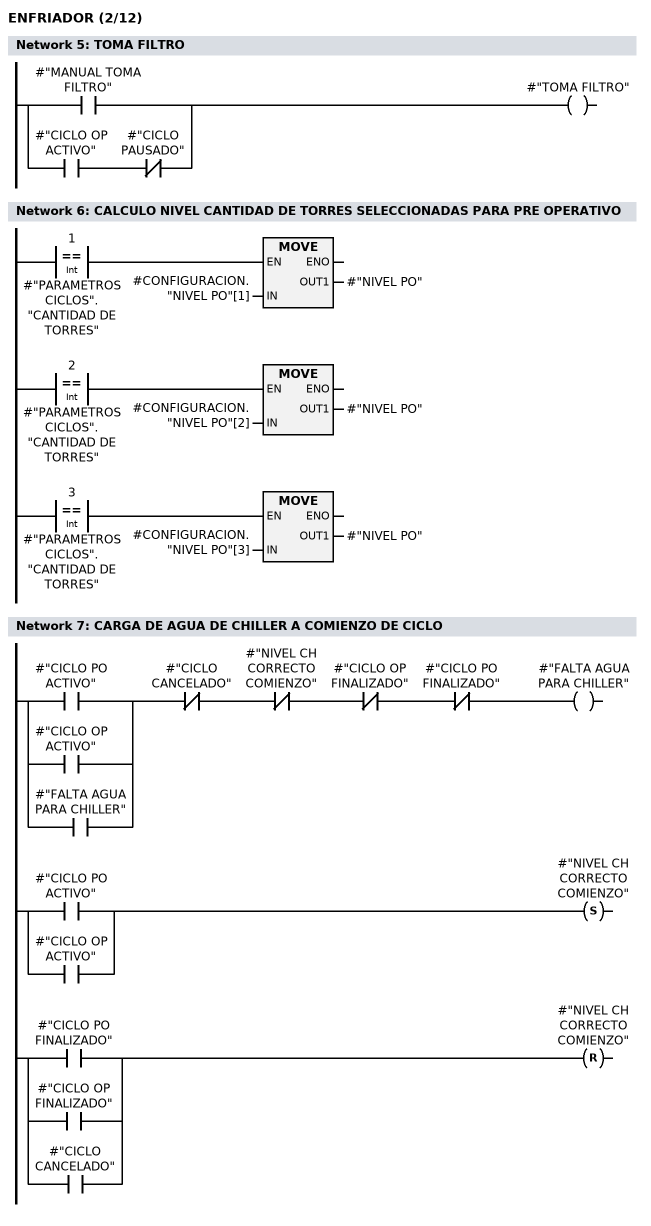
   RUNG wire#powerrail
      Contact( #"MANUAL TOMA FILTRO" )
      wire#w1
      Coil( #"TOMA FILTRO" )
   END_RUNG
   RUNG wire#powerrail
      Contact( #"CICLO OP ACTIVO" )
      I_Contact( #"CICLO PAUSADO" )
   END_RUNG wire#w1
   // the same network as SCL:
   #"TOMA FILTRO" := #"MANUAL TOMA FILTRO" OR (#"CICLO OP ACTIVO" AND NOT #"CICLO PAUSADO");
END_REGION

REGION Network 6: CALCULO NIVEL CANTIDAD DE TORRES SELECCIONADAS PARA PRE OPERATIVO
   RUNG wire#powerrail
      { S7_Templates := "SrcType := Int" } EQ_Contact(in1 := 1, in2 := #"PARAMETROS CICLOS"."CANTIDAD DE TORRES")
      Move(in := #CONFIGURACION."NIVEL PO"[1], out1 => #"NIVEL PO")
   END_RUNG
   RUNG wire#powerrail
      { S7_Templates := "SrcType := Int" } EQ_Contact(in1 := 2, in2 := #"PARAMETROS CICLOS"."CANTIDAD DE TORRES")
      Move(in := #CONFIGURACION."NIVEL PO"[2], out1 => #"NIVEL PO")
   END_RUNG
   RUNG wire#powerrail
      { S7_Templates := "SrcType := Int" } EQ_Contact(in1 := 3, in2 := #"PARAMETROS CICLOS"."CANTIDAD DE TORRES")
      Move(in := #CONFIGURACION."NIVEL PO"[3], out1 => #"NIVEL PO")
   END_RUNG
   // the same network as SCL:
   IF 1 = #"PARAMETROS CICLOS"."CANTIDAD DE TORRES" THEN #"NIVEL PO" := #CONFIGURACION."NIVEL PO"[1]; END_IF;
   IF 2 = #"PARAMETROS CICLOS"."CANTIDAD DE TORRES" THEN #"NIVEL PO" := #CONFIGURACION."NIVEL PO"[2]; END_IF;
   IF 3 = #"PARAMETROS CICLOS"."CANTIDAD DE TORRES" THEN #"NIVEL PO" := #CONFIGURACION."NIVEL PO"[3]; END_IF;
END_REGION

REGION Network 7: CARGA DE AGUA DE CHILLER A COMIENZO DE CICLO
   RUNG wire#powerrail
      Contact( #"CICLO PO ACTIVO" )
      wire#w1
      I_Contact( #"CICLO CANCELADO" )
      I_Contact( #"NIVEL CH CORRECTO COMIENZO" )
      I_Contact( #"CICLO OP FINALIZADO" )
      I_Contact( #"CICLO PO FINALIZADO" )
      Coil( #"FALTA AGUA PARA CHILLER" )
   END_RUNG
   RUNG wire#powerrail
      Contact( #"CICLO OP ACTIVO" )
   END_RUNG wire#w1
   RUNG wire#powerrail
      Contact( #"FALTA AGUA PARA CHILLER" )
   END_RUNG wire#w1
   RUNG wire#powerrail
      Contact( #"CICLO PO ACTIVO" )
      wire#w2
      S_Coil( #"NIVEL CH CORRECTO COMIENZO" )
   END_RUNG
   RUNG wire#powerrail
      Contact( #"CICLO OP ACTIVO" )
   END_RUNG wire#w2
   RUNG wire#powerrail
      Contact( #"CICLO PO FINALIZADO" )
      wire#w3
      R_Coil( #"NIVEL CH CORRECTO COMIENZO" )
   END_RUNG
   RUNG wire#powerrail
      Contact( #"CICLO OP FINALIZADO" )
   END_RUNG wire#w3
   RUNG wire#powerrail
      Contact( #"CICLO CANCELADO" )
   END_RUNG wire#w3
   // the same network as SCL:
   #"FALTA AGUA PARA CHILLER" := (#"CICLO PO ACTIVO" OR #"CICLO OP ACTIVO" OR #"FALTA AGUA PARA CHILLER") AND NOT #"CICLO CANCELADO" AND NOT #"NIVEL CH CORRECTO COMIENZO" AND NOT #"CICLO OP FINALIZADO" AND NOT #"CICLO PO FINALIZADO";
   IF #"CICLO PO ACTIVO" OR #"CICLO OP ACTIVO" THEN #"NIVEL CH CORRECTO COMIENZO" := TRUE; END_IF;
   IF #"CICLO PO FINALIZADO" OR #"CICLO OP FINALIZADO" OR #"CICLO CANCELADO" THEN
       #"NIVEL CH CORRECTO COMIENZO" := FALSE;
   END_IF;
END_REGION

REGION Network 8: CARGA DE AGUA PARA CHILLER VACIO
   // CARGAR AGUA TQ ( ABRIR VALVULA CARGA DE AGUA)
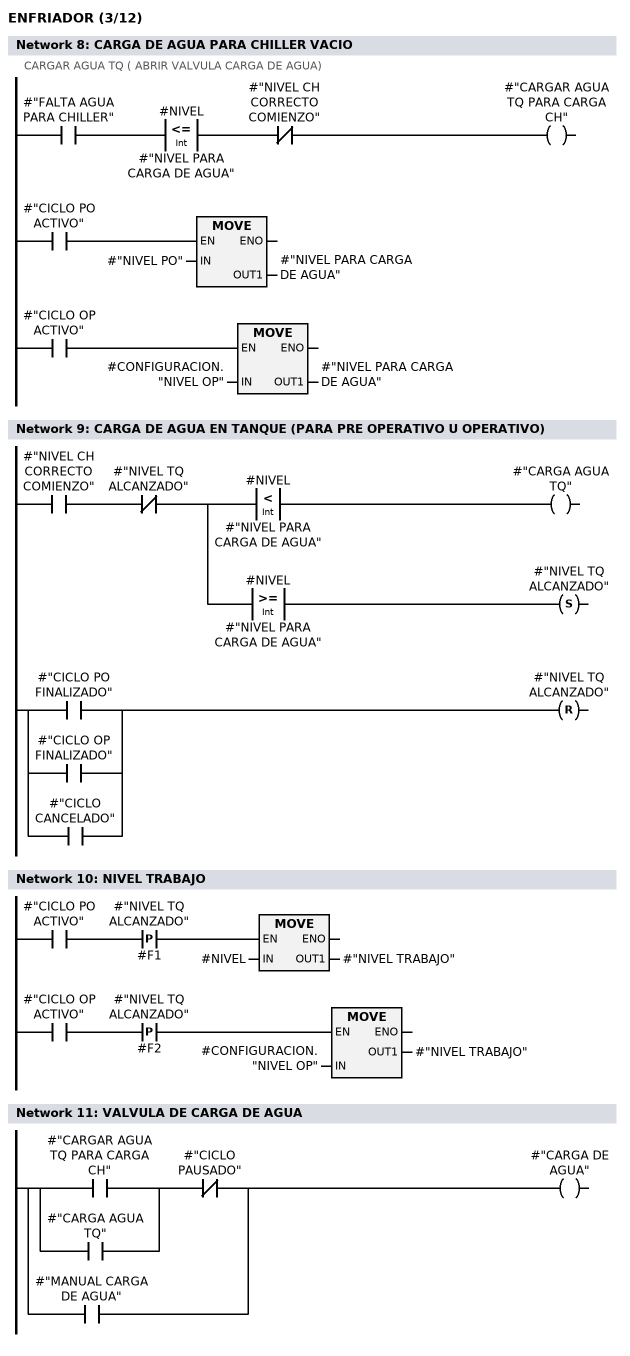
   RUNG wire#powerrail
      Contact( #"FALTA AGUA PARA CHILLER" )
      { S7_Templates := "SrcType := Int" } LE_Contact(in1 := #NIVEL, in2 := #"NIVEL PARA CARGA DE AGUA")
      I_Contact( #"NIVEL CH CORRECTO COMIENZO" )
      Coil( #"CARGAR AGUA TQ PARA CARGA CH" )
   END_RUNG
   RUNG wire#powerrail
      Contact( #"CICLO PO ACTIVO" )
      Move(in := #"NIVEL PO", out1 => #"NIVEL PARA CARGA DE AGUA")
   END_RUNG
   RUNG wire#powerrail
      Contact( #"CICLO OP ACTIVO" )
      Move(in := #CONFIGURACION."NIVEL OP", out1 => #"NIVEL PARA CARGA DE AGUA")
   END_RUNG
   // the same network as SCL:
   #"CARGAR AGUA TQ PARA CARGA CH" := #"FALTA AGUA PARA CHILLER" AND (#NIVEL <= #"NIVEL PARA CARGA DE AGUA") AND NOT #"NIVEL CH CORRECTO COMIENZO";
   IF #"CICLO PO ACTIVO" THEN #"NIVEL PARA CARGA DE AGUA" := #"NIVEL PO"; END_IF;
   IF #"CICLO OP ACTIVO" THEN #"NIVEL PARA CARGA DE AGUA" := #CONFIGURACION."NIVEL OP"; END_IF;
END_REGION

REGION Network 9: CARGA DE AGUA EN TANQUE (PARA PRE OPERATIVO U OPERATIVO)
   RUNG wire#powerrail
      Contact( #"NIVEL CH CORRECTO COMIENZO" )
      I_Contact( #"NIVEL TQ ALCANZADO" )
      wire#w1
      { S7_Templates := "SrcType := Int" } LT_Contact(in1 := #NIVEL, in2 := #"NIVEL PARA CARGA DE AGUA")
      Coil( #"CARGA AGUA TQ" )
   END_RUNG
   RUNG wire#w1
      { S7_Templates := "SrcType := Int" } GE_Contact(in1 := #NIVEL, in2 := #"NIVEL PARA CARGA DE AGUA")
      S_Coil( #"NIVEL TQ ALCANZADO" )
   END_RUNG
   RUNG wire#powerrail
      Contact( #"CICLO PO FINALIZADO" )
      wire#w2
      R_Coil( #"NIVEL TQ ALCANZADO" )
   END_RUNG
   RUNG wire#powerrail
      Contact( #"CICLO OP FINALIZADO" )
   END_RUNG wire#w2
   RUNG wire#powerrail
      Contact( #"CICLO CANCELADO" )
   END_RUNG wire#w2
   // the same network as SCL:
   #_w1 := #"NIVEL CH CORRECTO COMIENZO" AND NOT #"NIVEL TQ ALCANZADO";
   #"CARGA AGUA TQ" := #_w1 AND (#NIVEL < #"NIVEL PARA CARGA DE AGUA");
   IF #_w1 AND (#NIVEL >= #"NIVEL PARA CARGA DE AGUA") THEN #"NIVEL TQ ALCANZADO" := TRUE; END_IF;
   IF #"CICLO PO FINALIZADO" OR #"CICLO OP FINALIZADO" OR #"CICLO CANCELADO" THEN
       #"NIVEL TQ ALCANZADO" := FALSE;
   END_IF;
END_REGION

REGION Network 10: NIVEL TRABAJO
   RUNG wire#powerrail
      Contact( #"CICLO PO ACTIVO" )
      P_Contact(operand := #"NIVEL TQ ALCANZADO", bit := #F1)
      Move(in := #NIVEL, out1 => #"NIVEL TRABAJO")
   END_RUNG
   RUNG wire#powerrail
      Contact( #"CICLO OP ACTIVO" )
      P_Contact(operand := #"NIVEL TQ ALCANZADO", bit := #F2)
      Move(in := #CONFIGURACION."NIVEL OP", out1 => #"NIVEL TRABAJO")
   END_RUNG
   // the same network as SCL:
   #_w1 := #"CICLO PO ACTIVO" AND #"NIVEL TQ ALCANZADO" AND NOT #F1;   // rising edge of #"NIVEL TQ ALCANZADO"
   #F1 := #"NIVEL TQ ALCANZADO";
   IF #_w1 THEN #"NIVEL TRABAJO" := #NIVEL; END_IF;
   #_w2 := #"CICLO OP ACTIVO" AND #"NIVEL TQ ALCANZADO" AND NOT #F2;   // rising edge of #"NIVEL TQ ALCANZADO"
   #F2 := #"NIVEL TQ ALCANZADO";
   IF #_w2 THEN #"NIVEL TRABAJO" := #CONFIGURACION."NIVEL OP"; END_IF;
END_REGION

REGION Network 11: VALVULA DE CARGA DE AGUA
   RUNG wire#powerrail
      Contact( #"CARGAR AGUA TQ PARA CARGA CH" )
      wire#w1
      I_Contact( #"CICLO PAUSADO" )
      wire#w2
      Coil( #"CARGA DE AGUA" )
   END_RUNG
   RUNG wire#powerrail
      Contact( #"CARGA AGUA TQ" )
   END_RUNG wire#w1
   RUNG wire#powerrail
      Contact( #"MANUAL CARGA DE AGUA" )
   END_RUNG wire#w2
   // the same network as SCL:
   #"CARGA DE AGUA" := ((#"CARGAR AGUA TQ PARA CARGA CH" OR #"CARGA AGUA TQ") AND NOT #"CICLO PAUSADO") OR #"MANUAL CARGA DE AGUA";
END_REGION

REGION Network 12: MANDAR AGUA A CHILLER (CONTROL HISTERESIS DE NIVEL)
   // ENCENDIDO DE BOMBA DE EGRESO Y VALVULA (MANDAR AGUA A CHILLER)
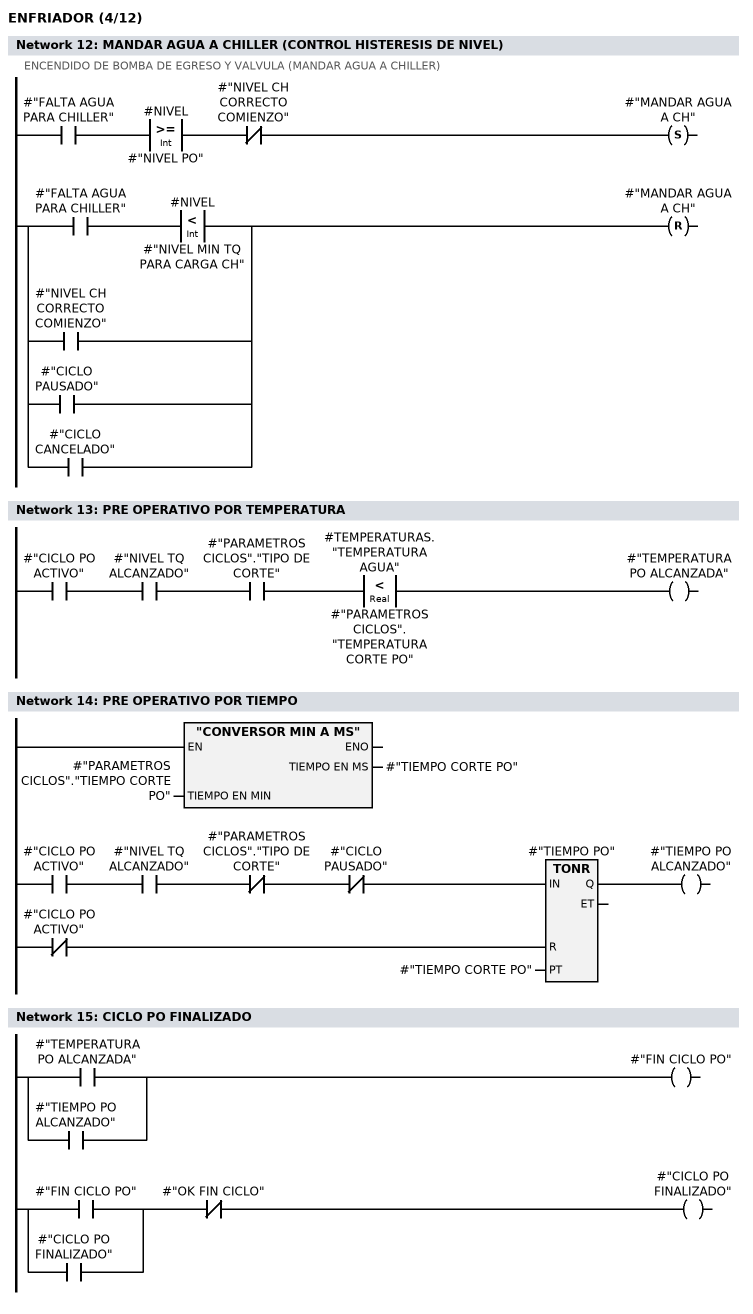
   RUNG wire#powerrail
      Contact( #"FALTA AGUA PARA CHILLER" )
      { S7_Templates := "SrcType := Int" } GE_Contact(in1 := #NIVEL, in2 := #"NIVEL PO")
      I_Contact( #"NIVEL CH CORRECTO COMIENZO" )
      S_Coil( #"MANDAR AGUA A CH" )
   END_RUNG
   RUNG wire#powerrail
      Contact( #"FALTA AGUA PARA CHILLER" )
      { S7_Templates := "SrcType := Int" } LT_Contact(in1 := #NIVEL, in2 := #"NIVEL MIN TQ PARA CARGA CH")
      wire#w1
      R_Coil( #"MANDAR AGUA A CH" )
   END_RUNG
   RUNG wire#powerrail
      Contact( #"NIVEL CH CORRECTO COMIENZO" )
   END_RUNG wire#w1
   RUNG wire#powerrail
      Contact( #"CICLO PAUSADO" )
   END_RUNG wire#w1
   RUNG wire#powerrail
      Contact( #"CICLO CANCELADO" )
   END_RUNG wire#w1
   // the same network as SCL:
   IF #"FALTA AGUA PARA CHILLER" AND (#NIVEL >= #"NIVEL PO") AND NOT #"NIVEL CH CORRECTO COMIENZO" THEN
       #"MANDAR AGUA A CH" := TRUE;
   END_IF;
   IF (#"FALTA AGUA PARA CHILLER" AND (#NIVEL < #"NIVEL MIN TQ PARA CARGA CH")) OR #"NIVEL CH CORRECTO COMIENZO" OR #"CICLO PAUSADO" OR #"CICLO CANCELADO" THEN
       #"MANDAR AGUA A CH" := FALSE;
   END_IF;
END_REGION

REGION Network 13: PRE OPERATIVO POR TEMPERATURA
   RUNG wire#powerrail
      Contact( #"CICLO PO ACTIVO" )
      Contact( #"NIVEL TQ ALCANZADO" )
      Contact( #"PARAMETROS CICLOS"."TIPO DE CORTE" )
      { S7_Templates := "SrcType := Real" } LT_Contact(in1 := #TEMPERATURAS."TEMPERATURA AGUA", in2 := #"PARAMETROS CICLOS"."TEMPERATURA CORTE PO")
      Coil( #"TEMPERATURA PO ALCANZADA" )
   END_RUNG
   // the same network as SCL:
   #"TEMPERATURA PO ALCANZADA" := #"CICLO PO ACTIVO" AND #"NIVEL TQ ALCANZADO" AND #"PARAMETROS CICLOS"."TIPO DE CORTE" AND (#TEMPERATURAS."TEMPERATURA AGUA" < #"PARAMETROS CICLOS"."TEMPERATURA CORTE PO");
END_REGION

REGION Network 14: PRE OPERATIVO POR TIEMPO
   "CONVERSOR MIN A MS"("TIEMPO EN MIN" := #"PARAMETROS CICLOS"."TIEMPO CORTE PO",
                        "TIEMPO EN MS" => #"TIEMPO CORTE PO");
   #"TIEMPO PO"(IN := #"CICLO PO ACTIVO" AND #"NIVEL TQ ALCANZADO" AND NOT #"PARAMETROS CICLOS"."TIPO DE CORTE" AND NOT #"CICLO PAUSADO",   // TONR
                R := NOT #"CICLO PO ACTIVO",
                PT := #"TIEMPO CORTE PO");
   #"TIEMPO PO ALCANZADO" := #"TIEMPO PO".Q;
END_REGION

REGION Network 15: CICLO PO FINALIZADO
   RUNG wire#powerrail
      Contact( #"TEMPERATURA PO ALCANZADA" )
      wire#w1
      Coil( #"FIN CICLO PO" )
   END_RUNG
   RUNG wire#powerrail
      Contact( #"TIEMPO PO ALCANZADO" )
   END_RUNG wire#w1
   RUNG wire#powerrail
      Contact( #"FIN CICLO PO" )
      wire#w2
      I_Contact( #"OK FIN CICLO" )
      Coil( #"CICLO PO FINALIZADO" )
   END_RUNG
   RUNG wire#powerrail
      Contact( #"CICLO PO FINALIZADO" )
   END_RUNG wire#w2
   // the same network as SCL:
   #"FIN CICLO PO" := #"TEMPERATURA PO ALCANZADA" OR #"TIEMPO PO ALCANZADO";
   #"CICLO PO FINALIZADO" := (#"FIN CICLO PO" OR #"CICLO PO FINALIZADO") AND NOT #"OK FIN CICLO";
END_REGION

REGION Network 16: INICIO CICLO OP
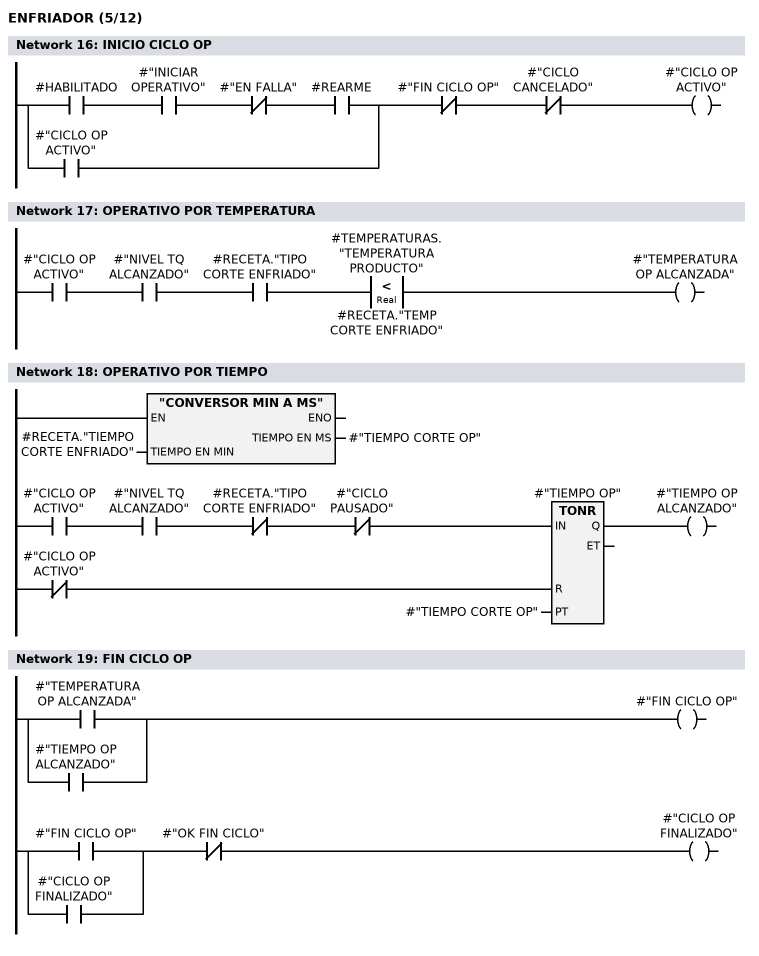
   RUNG wire#powerrail
      Contact( #HABILITADO )
      Contact( #"INICIAR OPERATIVO" )
      I_Contact( #"EN FALLA" )
      Contact( #REARME )
      wire#w1
      I_Contact( #"FIN CICLO OP" )
      I_Contact( #"CICLO CANCELADO" )
      Coil( #"CICLO OP ACTIVO" )
   END_RUNG
   RUNG wire#powerrail
      Contact( #"CICLO OP ACTIVO" )
   END_RUNG wire#w1
   // the same network as SCL:
   #"CICLO OP ACTIVO" := ((#HABILITADO AND #"INICIAR OPERATIVO" AND NOT #"EN FALLA" AND #REARME) OR #"CICLO OP ACTIVO") AND NOT #"FIN CICLO OP" AND NOT #"CICLO CANCELADO";
END_REGION

REGION Network 17: OPERATIVO POR TEMPERATURA
   RUNG wire#powerrail
      Contact( #"CICLO OP ACTIVO" )
      Contact( #"NIVEL TQ ALCANZADO" )
      Contact( #RECETA."TIPO CORTE ENFRIADO" )
      { S7_Templates := "SrcType := Real" } LT_Contact(in1 := #TEMPERATURAS."TEMPERATURA PRODUCTO", in2 := #RECETA."TEMP CORTE ENFRIADO")
      Coil( #"TEMPERATURA OP ALCANZADA" )
   END_RUNG
   // the same network as SCL:
   #"TEMPERATURA OP ALCANZADA" := #"CICLO OP ACTIVO" AND #"NIVEL TQ ALCANZADO" AND #RECETA."TIPO CORTE ENFRIADO" AND (#TEMPERATURAS."TEMPERATURA PRODUCTO" < #RECETA."TEMP CORTE ENFRIADO");
END_REGION

REGION Network 18: OPERATIVO POR TIEMPO
   "CONVERSOR MIN A MS"("TIEMPO EN MIN" := #RECETA."TIEMPO CORTE ENFRIADO",
                        "TIEMPO EN MS" => #"TIEMPO CORTE OP");
   #"TIEMPO OP"(IN := #"CICLO OP ACTIVO" AND #"NIVEL TQ ALCANZADO" AND NOT #RECETA."TIPO CORTE ENFRIADO" AND NOT #"CICLO PAUSADO",   // TONR
                R := NOT #"CICLO OP ACTIVO",
                PT := #"TIEMPO CORTE OP");
   #"TIEMPO OP ALCANZADO" := #"TIEMPO OP".Q;
END_REGION

REGION Network 19: FIN CICLO OP
   RUNG wire#powerrail
      Contact( #"TEMPERATURA OP ALCANZADA" )
      wire#w1
      Coil( #"FIN CICLO OP" )
   END_RUNG
   RUNG wire#powerrail
      Contact( #"TIEMPO OP ALCANZADO" )
   END_RUNG wire#w1
   RUNG wire#powerrail
      Contact( #"FIN CICLO OP" )
      wire#w2
      I_Contact( #"OK FIN CICLO" )
      Coil( #"CICLO OP FINALIZADO" )
   END_RUNG
   RUNG wire#powerrail
      Contact( #"CICLO OP FINALIZADO" )
   END_RUNG wire#w2
   // the same network as SCL:
   #"FIN CICLO OP" := #"TEMPERATURA OP ALCANZADA" OR #"TIEMPO OP ALCANZADO";
   #"CICLO OP FINALIZADO" := (#"FIN CICLO OP" OR #"CICLO OP FINALIZADO") AND NOT #"OK FIN CICLO";
END_REGION

REGION Network 20: CONTROL DE TEMPERATURA
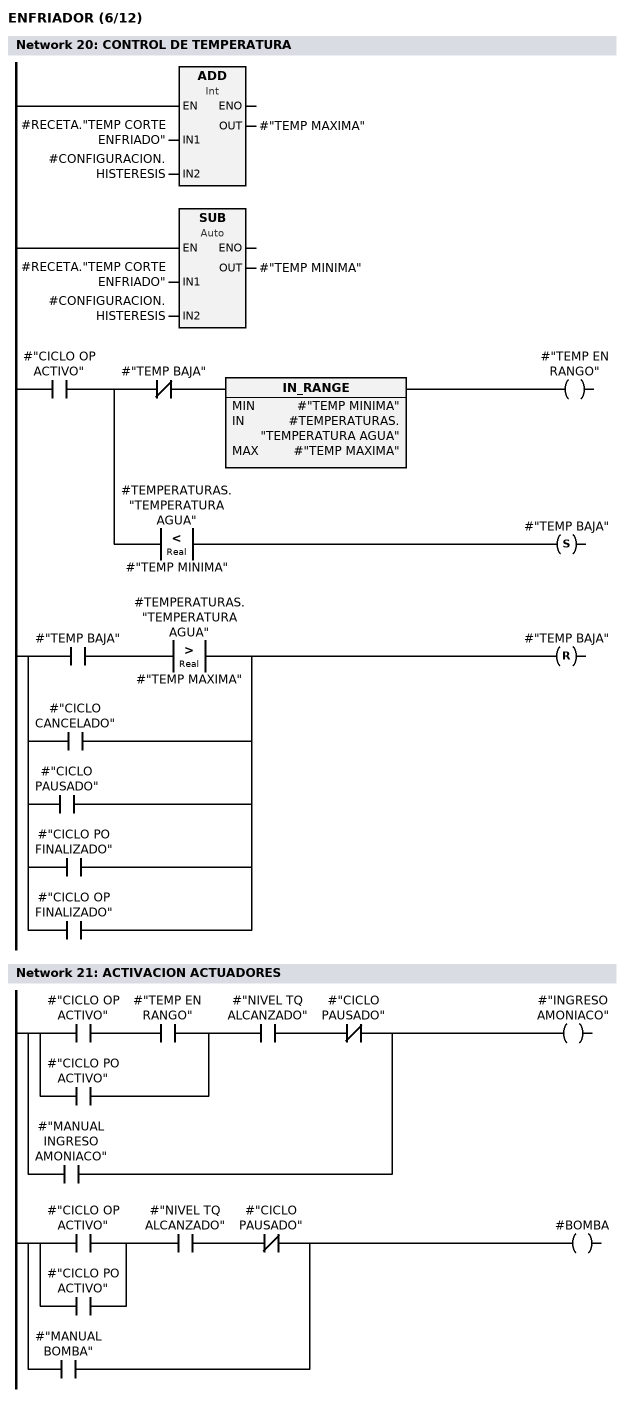
   RUNG wire#powerrail
      { S7_Templates := "SrcType := Int" } Add(in1 := #RECETA."TEMP CORTE ENFRIADO", in2 := #CONFIGURACION.HISTERESIS, out => #"TEMP MAXIMA")
   END_RUNG
   RUNG wire#powerrail
      Sub(in1 := #RECETA."TEMP CORTE ENFRIADO", in2 := #CONFIGURACION.HISTERESIS, out => #"TEMP MINIMA")
   END_RUNG
   RUNG wire#powerrail
      Contact( #"CICLO OP ACTIVO" )
      wire#w1
      I_Contact( #"TEMP BAJA" )
      { S7_Templates := "SrcType := Real" } InRange(min := #"TEMP MINIMA", in := #TEMPERATURAS."TEMPERATURA AGUA", max := #"TEMP MAXIMA")
      Coil( #"TEMP EN RANGO" )
   END_RUNG
   RUNG wire#w1
      { S7_Templates := "SrcType := Real" } LT_Contact(in1 := #TEMPERATURAS."TEMPERATURA AGUA", in2 := #"TEMP MINIMA")
      S_Coil( #"TEMP BAJA" )
   END_RUNG
   RUNG wire#powerrail
      Contact( #"TEMP BAJA" )
      { S7_Templates := "SrcType := Real" } GT_Contact(in1 := #TEMPERATURAS."TEMPERATURA AGUA", in2 := #"TEMP MAXIMA")
      wire#w2
      R_Coil( #"TEMP BAJA" )
   END_RUNG
   RUNG wire#powerrail
      Contact( #"CICLO CANCELADO" )
   END_RUNG wire#w2
   RUNG wire#powerrail
      Contact( #"CICLO PAUSADO" )
   END_RUNG wire#w2
   RUNG wire#powerrail
      Contact( #"CICLO PO FINALIZADO" )
   END_RUNG wire#w2
   RUNG wire#powerrail
      Contact( #"CICLO OP FINALIZADO" )
   END_RUNG wire#w2
   // the same network as SCL:
   #"TEMP MAXIMA" := #RECETA."TEMP CORTE ENFRIADO" + #CONFIGURACION.HISTERESIS;
   #"TEMP MINIMA" := #RECETA."TEMP CORTE ENFRIADO" - #CONFIGURACION.HISTERESIS;
   #"TEMP EN RANGO" := #"CICLO OP ACTIVO" AND NOT #"TEMP BAJA" AND (#"TEMP MINIMA" <= #TEMPERATURAS."TEMPERATURA AGUA") AND (#TEMPERATURAS."TEMPERATURA AGUA" <= #"TEMP MAXIMA");
   IF #"CICLO OP ACTIVO" AND (#TEMPERATURAS."TEMPERATURA AGUA" < #"TEMP MINIMA") THEN
       #"TEMP BAJA" := TRUE;
   END_IF;
   IF (#"TEMP BAJA" AND (#TEMPERATURAS."TEMPERATURA AGUA" > #"TEMP MAXIMA")) OR #"CICLO CANCELADO" OR #"CICLO PAUSADO" OR #"CICLO PO FINALIZADO" OR #"CICLO OP FINALIZADO" THEN
       #"TEMP BAJA" := FALSE;
   END_IF;
END_REGION

REGION Network 21: ACTIVACION ACTUADORES
   RUNG wire#powerrail
      Contact( #"CICLO OP ACTIVO" )
      Contact( #"TEMP EN RANGO" )
      wire#w1
      Contact( #"NIVEL TQ ALCANZADO" )
      I_Contact( #"CICLO PAUSADO" )
      wire#w2
      Coil( #"INGRESO AMONIACO" )
   END_RUNG
   RUNG wire#powerrail
      Contact( #"CICLO PO ACTIVO" )
   END_RUNG wire#w1
   RUNG wire#powerrail
      Contact( #"MANUAL INGRESO AMONIACO" )
   END_RUNG wire#w2
   RUNG wire#powerrail
      Contact( #"CICLO OP ACTIVO" )
      wire#w3
      Contact( #"NIVEL TQ ALCANZADO" )
      I_Contact( #"CICLO PAUSADO" )
      wire#w4
      Coil( #BOMBA )
   END_RUNG
   RUNG wire#powerrail
      Contact( #"CICLO PO ACTIVO" )
   END_RUNG wire#w3
   RUNG wire#powerrail
      Contact( #"MANUAL BOMBA" )
   END_RUNG wire#w4
   // the same network as SCL:
   #"INGRESO AMONIACO" := (((#"CICLO OP ACTIVO" AND #"TEMP EN RANGO") OR #"CICLO PO ACTIVO") AND #"NIVEL TQ ALCANZADO" AND NOT #"CICLO PAUSADO") OR #"MANUAL INGRESO AMONIACO";
   #BOMBA := ((#"CICLO OP ACTIVO" OR #"CICLO PO ACTIVO") AND #"NIVEL TQ ALCANZADO" AND NOT #"CICLO PAUSADO") OR #"MANUAL BOMBA";
END_REGION

REGION Network 22: ESTADO EQUIPO (COLOR HMI EN PRINCIPAL)
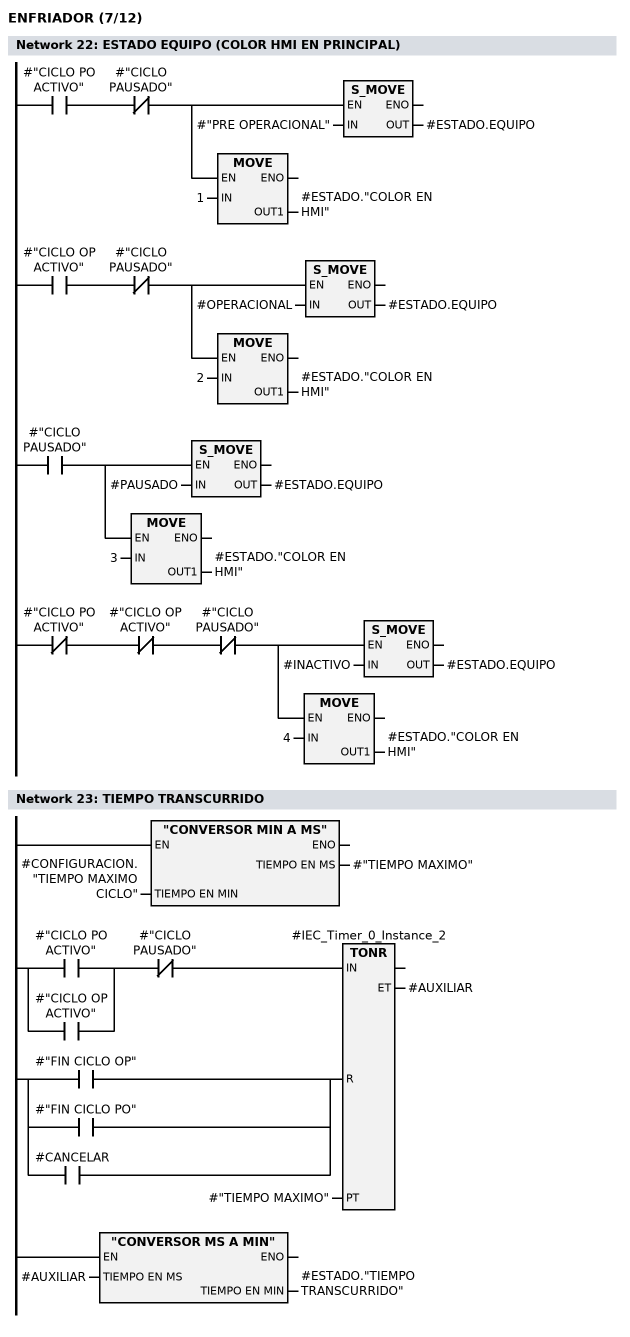
   RUNG wire#powerrail
      Contact( #"CICLO PO ACTIVO" )
      I_Contact( #"CICLO PAUSADO" )
      wire#w1
      S_Move(in := #"PRE OPERACIONAL", out => #ESTADO.EQUIPO)
   END_RUNG
   RUNG wire#w1
      Move(in := 1, out1 => #ESTADO."COLOR EN HMI")
   END_RUNG
   RUNG wire#powerrail
      Contact( #"CICLO OP ACTIVO" )
      I_Contact( #"CICLO PAUSADO" )
      wire#w2
      S_Move(in := #OPERACIONAL, out => #ESTADO.EQUIPO)
   END_RUNG
   RUNG wire#w2
      Move(in := 2, out1 => #ESTADO."COLOR EN HMI")
   END_RUNG
   RUNG wire#powerrail
      Contact( #"CICLO PAUSADO" )
      wire#w3
      S_Move(in := #PAUSADO, out => #ESTADO.EQUIPO)
   END_RUNG
   RUNG wire#w3
      Move(in := 3, out1 => #ESTADO."COLOR EN HMI")
   END_RUNG
   RUNG wire#powerrail
      I_Contact( #"CICLO PO ACTIVO" )
      I_Contact( #"CICLO OP ACTIVO" )
      I_Contact( #"CICLO PAUSADO" )
      wire#w4
      S_Move(in := #INACTIVO, out => #ESTADO.EQUIPO)
   END_RUNG
   RUNG wire#w4
      Move(in := 4, out1 => #ESTADO."COLOR EN HMI")
   END_RUNG
   // the same network as SCL:
   IF #"CICLO PO ACTIVO" AND NOT #"CICLO PAUSADO" THEN
       #ESTADO.EQUIPO := #"PRE OPERACIONAL";
       #ESTADO."COLOR EN HMI" := 1;
   END_IF;
   IF #"CICLO OP ACTIVO" AND NOT #"CICLO PAUSADO" THEN
       #ESTADO.EQUIPO := #OPERACIONAL;
       #ESTADO."COLOR EN HMI" := 2;
   END_IF;
   IF #"CICLO PAUSADO" THEN
       #ESTADO.EQUIPO := #PAUSADO;
       #ESTADO."COLOR EN HMI" := 3;
   END_IF;
   IF NOT #"CICLO PO ACTIVO" AND NOT #"CICLO OP ACTIVO" AND NOT #"CICLO PAUSADO" THEN
       #ESTADO.EQUIPO := #INACTIVO;
       #ESTADO."COLOR EN HMI" := 4;
   END_IF;
END_REGION

REGION Network 23: TIEMPO TRANSCURRIDO
   "CONVERSOR MIN A MS"("TIEMPO EN MIN" := #CONFIGURACION."TIEMPO MAXIMO CICLO",
                        "TIEMPO EN MS" => #"TIEMPO MAXIMO");
   #IEC_Timer_0_Instance_2(IN := (#"CICLO PO ACTIVO" OR #"CICLO OP ACTIVO") AND NOT #"CICLO PAUSADO",   // TONR
                           R := #"FIN CICLO OP" OR #"FIN CICLO PO" OR #CANCELAR,
                           PT := #"TIEMPO MAXIMO",
                           ET => #AUXILIAR);
   "CONVERSOR MS A MIN"("TIEMPO EN MS" := #AUXILIAR, "TIEMPO EN MIN" => #ESTADO."TIEMPO TRANSCURRIDO");
END_REGION

REGION Network 24: VISIBILIDAD HMI ************* MODIFICACION EN ESTADO EN CICLO
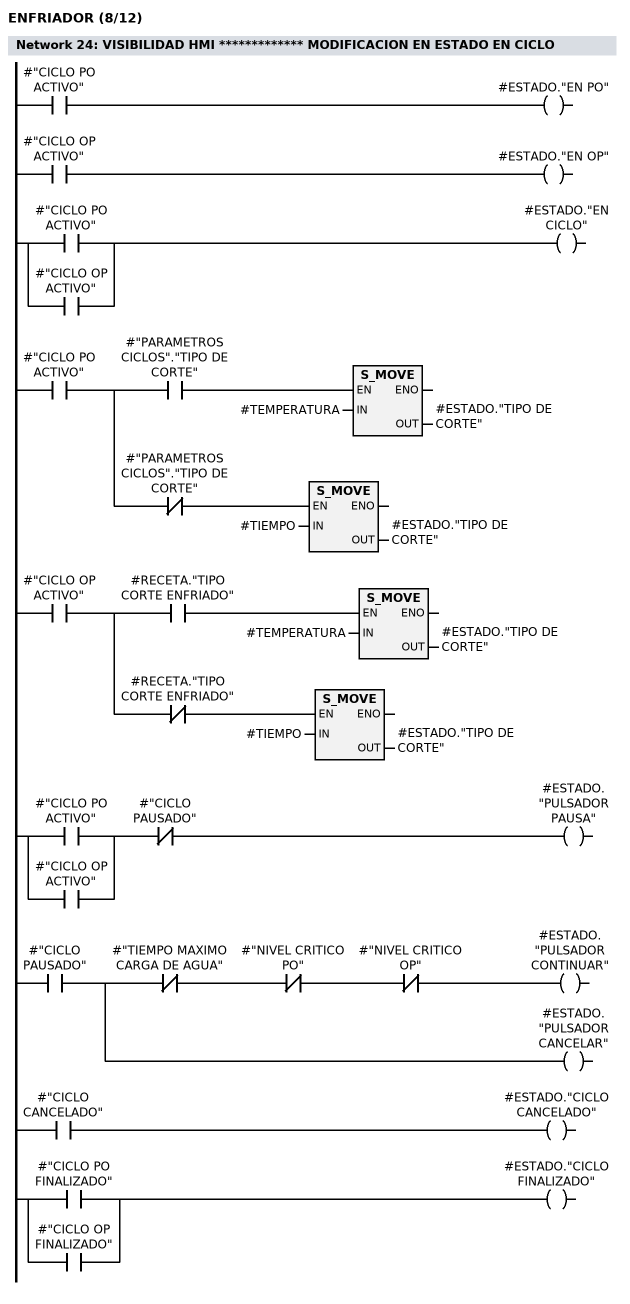
   RUNG wire#powerrail
      Contact( #"CICLO PO ACTIVO" )
      Coil( #ESTADO."EN PO" )
   END_RUNG
   RUNG wire#powerrail
      Contact( #"CICLO OP ACTIVO" )
      Coil( #ESTADO."EN OP" )
   END_RUNG
   RUNG wire#powerrail
      Contact( #"CICLO PO ACTIVO" )
      wire#w1
      Coil( #ESTADO."EN CICLO" )
   END_RUNG
   RUNG wire#powerrail
      Contact( #"CICLO OP ACTIVO" )
   END_RUNG wire#w1
   RUNG wire#powerrail
      Contact( #"CICLO PO ACTIVO" )
      wire#w2
      Contact( #"PARAMETROS CICLOS"."TIPO DE CORTE" )
      S_Move(in := #TEMPERATURA, out => #ESTADO."TIPO DE CORTE")
   END_RUNG
   RUNG wire#w2
      I_Contact( #"PARAMETROS CICLOS"."TIPO DE CORTE" )
      S_Move(in := #TIEMPO, out => #ESTADO."TIPO DE CORTE")
   END_RUNG
   RUNG wire#powerrail
      Contact( #"CICLO OP ACTIVO" )
      wire#w3
      Contact( #RECETA."TIPO CORTE ENFRIADO" )
      S_Move(in := #TEMPERATURA, out => #ESTADO."TIPO DE CORTE")
   END_RUNG
   RUNG wire#w3
      I_Contact( #RECETA."TIPO CORTE ENFRIADO" )
      S_Move(in := #TIEMPO, out => #ESTADO."TIPO DE CORTE")
   END_RUNG
   RUNG wire#powerrail
      Contact( #"CICLO PO ACTIVO" )
      wire#w4
      I_Contact( #"CICLO PAUSADO" )
      Coil( #ESTADO."PULSADOR PAUSA" )
   END_RUNG
   RUNG wire#powerrail
      Contact( #"CICLO OP ACTIVO" )
   END_RUNG wire#w4
   RUNG wire#powerrail
      Contact( #"CICLO PAUSADO" )
      wire#w5
      I_Contact( #"TIEMPO MAXIMO CARGA DE AGUA" )
      I_Contact( #"NIVEL CRITICO PO" )
      I_Contact( #"NIVEL CRITICO OP" )
      Coil( #ESTADO."PULSADOR CONTINUAR" )
   END_RUNG
   RUNG wire#w5
      Coil( #ESTADO."PULSADOR CANCELAR" )
   END_RUNG
   RUNG wire#powerrail
      Contact( #"CICLO CANCELADO" )
      Coil( #ESTADO."CICLO CANCELADO" )
   END_RUNG
   RUNG wire#powerrail
      Contact( #"CICLO PO FINALIZADO" )
      wire#w6
      Coil( #ESTADO."CICLO FINALIZADO" )
   END_RUNG
   RUNG wire#powerrail
      Contact( #"CICLO OP FINALIZADO" )
   END_RUNG wire#w6
   // the same network as SCL:
   #ESTADO."EN PO" := #"CICLO PO ACTIVO";
   #ESTADO."EN OP" := #"CICLO OP ACTIVO";
   #ESTADO."EN CICLO" := #"CICLO PO ACTIVO" OR #"CICLO OP ACTIVO";
   IF #"CICLO PO ACTIVO" AND #"PARAMETROS CICLOS"."TIPO DE CORTE" THEN
       #ESTADO."TIPO DE CORTE" := #TEMPERATURA;
   END_IF;
   IF #"CICLO PO ACTIVO" AND NOT #"PARAMETROS CICLOS"."TIPO DE CORTE" THEN
       #ESTADO."TIPO DE CORTE" := #TIEMPO;
   END_IF;
   IF #"CICLO OP ACTIVO" AND #RECETA."TIPO CORTE ENFRIADO" THEN
       #ESTADO."TIPO DE CORTE" := #TEMPERATURA;
   END_IF;
   IF #"CICLO OP ACTIVO" AND NOT #RECETA."TIPO CORTE ENFRIADO" THEN
       #ESTADO."TIPO DE CORTE" := #TIEMPO;
   END_IF;
   #ESTADO."PULSADOR PAUSA" := (#"CICLO PO ACTIVO" OR #"CICLO OP ACTIVO") AND NOT #"CICLO PAUSADO";
   #ESTADO."PULSADOR CONTINUAR" := #"CICLO PAUSADO" AND NOT #"TIEMPO MAXIMO CARGA DE AGUA" AND NOT #"NIVEL CRITICO PO" AND NOT #"NIVEL CRITICO OP";
   #ESTADO."PULSADOR CANCELAR" := #"CICLO PAUSADO";
   #ESTADO."CICLO CANCELADO" := #"CICLO CANCELADO";
   #ESTADO."CICLO FINALIZADO" := #"CICLO PO FINALIZADO" OR #"CICLO OP FINALIZADO";
END_REGION

REGION Network 25: RESET ACTUADORES MANUAL
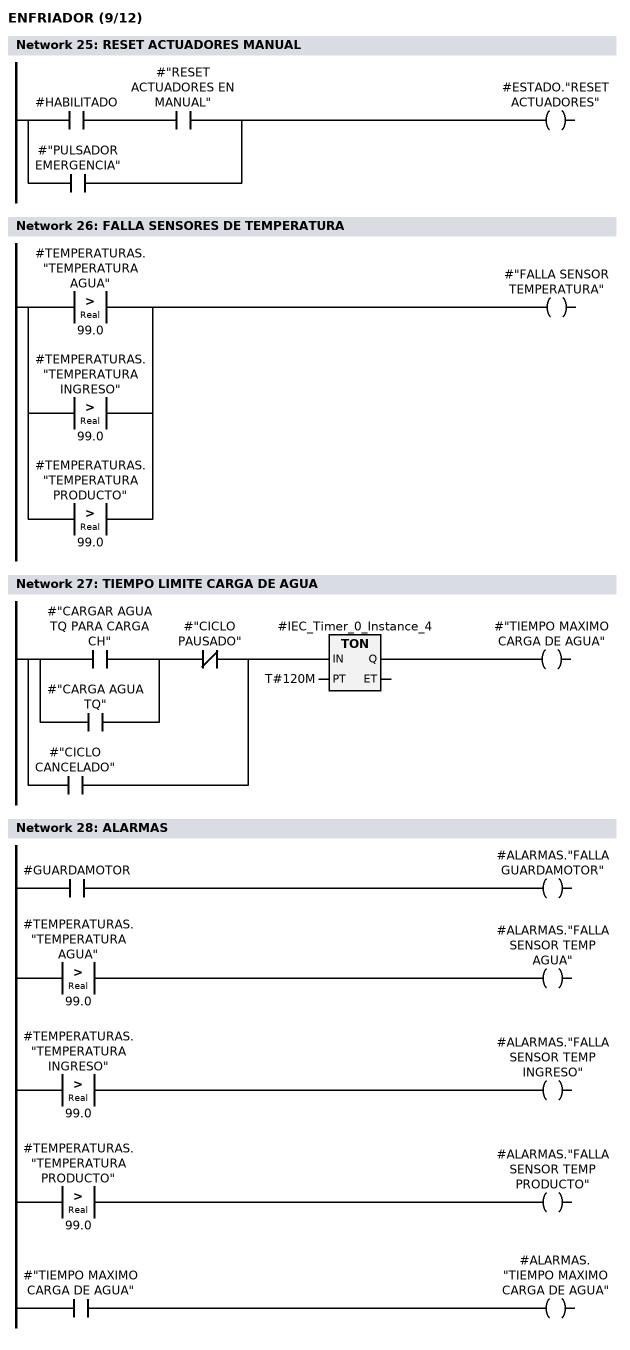
   RUNG wire#powerrail
      Contact( #HABILITADO )
      Contact( #"RESET ACTUADORES EN MANUAL" )
      wire#w1
      Coil( #ESTADO."RESET ACTUADORES" )
   END_RUNG
   RUNG wire#powerrail
      Contact( #"PULSADOR EMERGENCIA" )
   END_RUNG wire#w1
   // the same network as SCL:
   #ESTADO."RESET ACTUADORES" := (#HABILITADO AND #"RESET ACTUADORES EN MANUAL") OR #"PULSADOR EMERGENCIA";
END_REGION

REGION Network 26: FALLA SENSORES DE TEMPERATURA
   RUNG wire#powerrail
      { S7_Templates := "SrcType := Real" } GT_Contact(in1 := #TEMPERATURAS."TEMPERATURA AGUA", in2 := 99.0)
      wire#w1
      Coil( #"FALLA SENSOR TEMPERATURA" )
   END_RUNG
   RUNG wire#powerrail
      { S7_Templates := "SrcType := Real" } GT_Contact(in1 := #TEMPERATURAS."TEMPERATURA INGRESO", in2 := 99.0)
   END_RUNG wire#w1
   RUNG wire#powerrail
      { S7_Templates := "SrcType := Real" } GT_Contact(in1 := #TEMPERATURAS."TEMPERATURA PRODUCTO", in2 := 99.0)
   END_RUNG wire#w1
   // the same network as SCL:
   #"FALLA SENSOR TEMPERATURA" := (#TEMPERATURAS."TEMPERATURA AGUA" > 99.0) OR (#TEMPERATURAS."TEMPERATURA INGRESO" > 99.0) OR (#TEMPERATURAS."TEMPERATURA PRODUCTO" > 99.0);
END_REGION

REGION Network 27: TIEMPO LIMITE CARGA DE AGUA
   #IEC_Timer_0_Instance_4(IN := ((#"CARGAR AGUA TQ PARA CARGA CH" OR #"CARGA AGUA TQ") AND NOT #"CICLO PAUSADO") OR #"CICLO CANCELADO",   // TON
                           PT := T#120M);
   #"TIEMPO MAXIMO CARGA DE AGUA" := #IEC_Timer_0_Instance_4.Q;
END_REGION

REGION Network 28: ALARMAS
   RUNG wire#powerrail
      Contact( #GUARDAMOTOR )
      Coil( #ALARMAS."FALLA GUARDAMOTOR" )
   END_RUNG
   RUNG wire#powerrail
      { S7_Templates := "SrcType := Real" } GT_Contact(in1 := #TEMPERATURAS."TEMPERATURA AGUA", in2 := 99.0)
      Coil( #ALARMAS."FALLA SENSOR TEMP AGUA" )
   END_RUNG
   RUNG wire#powerrail
      { S7_Templates := "SrcType := Real" } GT_Contact(in1 := #TEMPERATURAS."TEMPERATURA INGRESO", in2 := 99.0)
      Coil( #ALARMAS."FALLA SENSOR TEMP INGRESO" )
   END_RUNG
   RUNG wire#powerrail
      { S7_Templates := "SrcType := Real" } GT_Contact(in1 := #TEMPERATURAS."TEMPERATURA PRODUCTO", in2 := 99.0)
      Coil( #ALARMAS."FALLA SENSOR TEMP PRODUCTO" )
   END_RUNG
   RUNG wire#powerrail
      Contact( #"TIEMPO MAXIMO CARGA DE AGUA" )
      Coil( #ALARMAS."TIEMPO MAXIMO CARGA DE AGUA" )
   END_RUNG
   // the same network as SCL:
   #ALARMAS."FALLA GUARDAMOTOR" := #GUARDAMOTOR;
   #ALARMAS."FALLA SENSOR TEMP AGUA" := #TEMPERATURAS."TEMPERATURA AGUA" > 99.0;
   #ALARMAS."FALLA SENSOR TEMP INGRESO" := #TEMPERATURAS."TEMPERATURA INGRESO" > 99.0;
   #ALARMAS."FALLA SENSOR TEMP PRODUCTO" := #TEMPERATURAS."TEMPERATURA PRODUCTO" > 99.0;
   #ALARMAS."TIEMPO MAXIMO CARGA DE AGUA" := #"TIEMPO MAXIMO CARGA DE AGUA";
END_REGION

REGION Network 29: ACTUADORES EN MODO MANUAL ACTIVOS
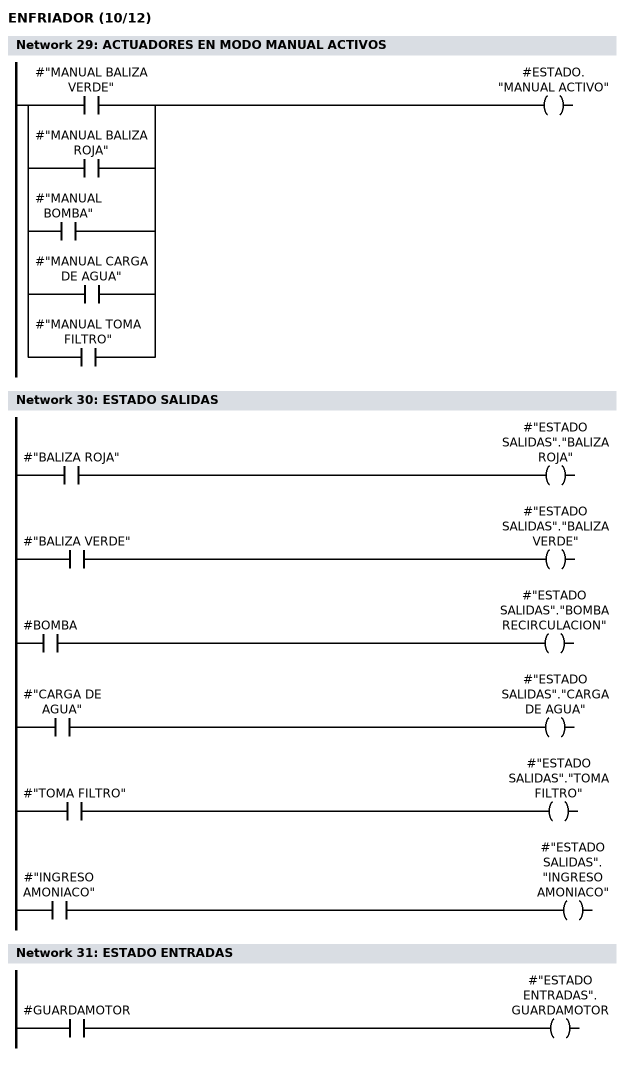
   RUNG wire#powerrail
      Contact( #"MANUAL BALIZA VERDE" )
      wire#w1
      Coil( #ESTADO."MANUAL ACTIVO" )
   END_RUNG
   RUNG wire#powerrail
      Contact( #"MANUAL BALIZA ROJA" )
   END_RUNG wire#w1
   RUNG wire#powerrail
      Contact( #"MANUAL BOMBA" )
   END_RUNG wire#w1
   RUNG wire#powerrail
      Contact( #"MANUAL CARGA DE AGUA" )
   END_RUNG wire#w1
   RUNG wire#powerrail
      Contact( #"MANUAL TOMA FILTRO" )
   END_RUNG wire#w1
   // the same network as SCL:
   #ESTADO."MANUAL ACTIVO" := #"MANUAL BALIZA VERDE" OR #"MANUAL BALIZA ROJA" OR #"MANUAL BOMBA" OR #"MANUAL CARGA DE AGUA" OR #"MANUAL TOMA FILTRO";
END_REGION

REGION Network 30: ESTADO SALIDAS
   RUNG wire#powerrail
      Contact( #"BALIZA ROJA" )
      Coil( #"ESTADO SALIDAS"."BALIZA ROJA" )
   END_RUNG
   RUNG wire#powerrail
      Contact( #"BALIZA VERDE" )
      Coil( #"ESTADO SALIDAS"."BALIZA VERDE" )
   END_RUNG
   RUNG wire#powerrail
      Contact( #BOMBA )
      Coil( #"ESTADO SALIDAS"."BOMBA RECIRCULACION" )
   END_RUNG
   RUNG wire#powerrail
      Contact( #"CARGA DE AGUA" )
      Coil( #"ESTADO SALIDAS"."CARGA DE AGUA" )
   END_RUNG
   RUNG wire#powerrail
      Contact( #"TOMA FILTRO" )
      Coil( #"ESTADO SALIDAS"."TOMA FILTRO" )
   END_RUNG
   RUNG wire#powerrail
      Contact( #"INGRESO AMONIACO" )
      Coil( #"ESTADO SALIDAS"."INGRESO AMONIACO" )
   END_RUNG
   // the same network as SCL:
   #"ESTADO SALIDAS"."BALIZA ROJA" := #"BALIZA ROJA";
   #"ESTADO SALIDAS"."BALIZA VERDE" := #"BALIZA VERDE";
   #"ESTADO SALIDAS"."BOMBA RECIRCULACION" := #BOMBA;
   #"ESTADO SALIDAS"."CARGA DE AGUA" := #"CARGA DE AGUA";
   #"ESTADO SALIDAS"."TOMA FILTRO" := #"TOMA FILTRO";
   #"ESTADO SALIDAS"."INGRESO AMONIACO" := #"INGRESO AMONIACO";
END_REGION

REGION Network 31: ESTADO ENTRADAS
   RUNG wire#powerrail
      Contact( #GUARDAMOTOR )
      Coil( #"ESTADO ENTRADAS".GUARDAMOTOR )
   END_RUNG
   // the same network as SCL:
   #"ESTADO ENTRADAS".GUARDAMOTOR := #GUARDAMOTOR;
END_REGION

REGION Network 32: NIVELES CRITICOS
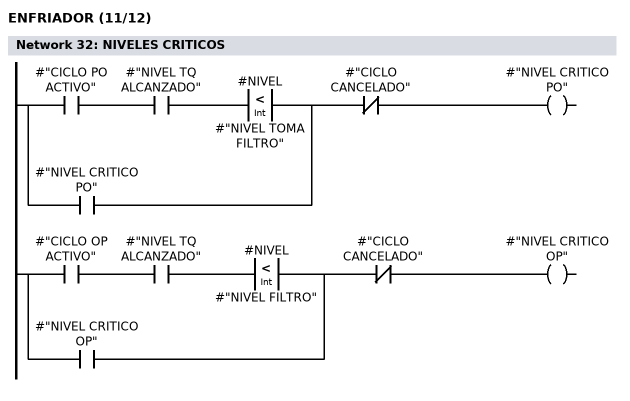
   RUNG wire#powerrail
      Contact( #"CICLO PO ACTIVO" )
      Contact( #"NIVEL TQ ALCANZADO" )
      { S7_Templates := "SrcType := Int" } LT_Contact(in1 := #NIVEL, in2 := #"NIVEL TOMA FILTRO")
      wire#w1
      I_Contact( #"CICLO CANCELADO" )
      Coil( #"NIVEL CRITICO PO" )
   END_RUNG
   RUNG wire#powerrail
      Contact( #"NIVEL CRITICO PO" )
   END_RUNG wire#w1
   RUNG wire#powerrail
      Contact( #"CICLO OP ACTIVO" )
      Contact( #"NIVEL TQ ALCANZADO" )
      { S7_Templates := "SrcType := Int" } LT_Contact(in1 := #NIVEL, in2 := #"NIVEL FILTRO")
      wire#w2
      I_Contact( #"CICLO CANCELADO" )
      Coil( #"NIVEL CRITICO OP" )
   END_RUNG
   RUNG wire#powerrail
      Contact( #"NIVEL CRITICO OP" )
   END_RUNG wire#w2
   // the same network as SCL:
   #"NIVEL CRITICO PO" := ((#"CICLO PO ACTIVO" AND #"NIVEL TQ ALCANZADO" AND (#NIVEL < #"NIVEL TOMA FILTRO")) OR #"NIVEL CRITICO PO") AND NOT #"CICLO CANCELADO";
   #"NIVEL CRITICO OP" := ((#"CICLO OP ACTIVO" AND #"NIVEL TQ ALCANZADO" AND (#NIVEL < #"NIVEL FILTRO")) OR #"NIVEL CRITICO OP") AND NOT #"CICLO CANCELADO";
END_REGION

REGION Network 33: SEÑALIZACIONES
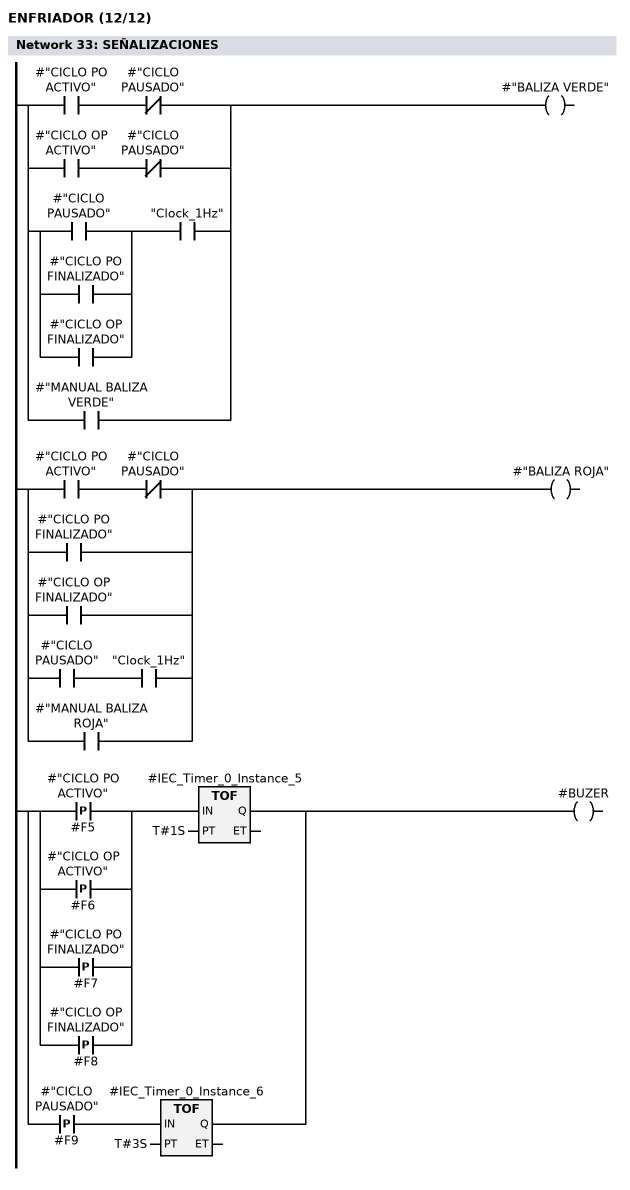
   #"BALIZA VERDE" := (#"CICLO PO ACTIVO" AND NOT #"CICLO PAUSADO") OR (#"CICLO OP ACTIVO" AND NOT #"CICLO PAUSADO") OR ((#"CICLO PAUSADO" OR #"CICLO PO FINALIZADO" OR #"CICLO OP FINALIZADO") AND "Clock_1Hz") OR #"MANUAL BALIZA VERDE";
   #"BALIZA ROJA" := (#"CICLO PO ACTIVO" AND NOT #"CICLO PAUSADO") OR #"CICLO PO FINALIZADO" OR #"CICLO OP FINALIZADO" OR (#"CICLO PAUSADO" AND "Clock_1Hz") OR #"MANUAL BALIZA ROJA";
   #_w1 := #"CICLO PO ACTIVO" AND NOT #F5;   // rising edge of #"CICLO PO ACTIVO"
   #F5 := #"CICLO PO ACTIVO";
   #_w2 := #"CICLO OP ACTIVO" AND NOT #F6;   // rising edge of #"CICLO OP ACTIVO"
   #F6 := #"CICLO OP ACTIVO";
   #_w3 := #"CICLO PO FINALIZADO" AND NOT #F7;   // rising edge of #"CICLO PO FINALIZADO"
   #F7 := #"CICLO PO FINALIZADO";
   #_w4 := #"CICLO OP FINALIZADO" AND NOT #F8;   // rising edge of #"CICLO OP FINALIZADO"
   #F8 := #"CICLO OP FINALIZADO";
   #IEC_Timer_0_Instance_5(IN := #_w1 OR #_w2 OR #_w3 OR #_w4, PT := T#1S);   // TOF
   #_w5 := #"CICLO PAUSADO" AND NOT #F9;   // rising edge of #"CICLO PAUSADO"
   #F9 := #"CICLO PAUSADO";
   #IEC_Timer_0_Instance_6(IN := #_w5, PT := T#3S);   // TOF
   #BUZER := #IEC_Timer_0_Instance_5.Q OR #IEC_Timer_0_Instance_6.Q;
END_REGION
END_FUNCTION_BLOCK

FUNCTION_BLOCK "SELECCION DE EQUIPO"   // FB2, LAD
{ S7_Optimized_Access := 'TRUE' }
VERSION : 0.1
   VAR_INPUT
      "AUMENTAR EQUIPO" : Bool;
      "DISMINUIR EQUIPO" : Bool;
      "VER EQUIPO 1" : Bool;
      "VER EQUIPO 2" : Bool;
   END_VAR
   VAR_OUTPUT
      "EQUIPO SELECCIONADO" : Int;
      "ACTUALIZAR EQUIPO" : Bool;
   END_VAR
   VAR RETAIN
      IEC_Counter_0_Instance : CTUD_INT;
      "IR A NUMERO DE EQUIPO SELECCIONADO" : Bool;
   END_VAR
   VAR
      "NUMERO DE EQUIPO ELEGIDO" : Int;
      AUXILIAR : Int;
   END_VAR
BEGIN

REGION Network 1
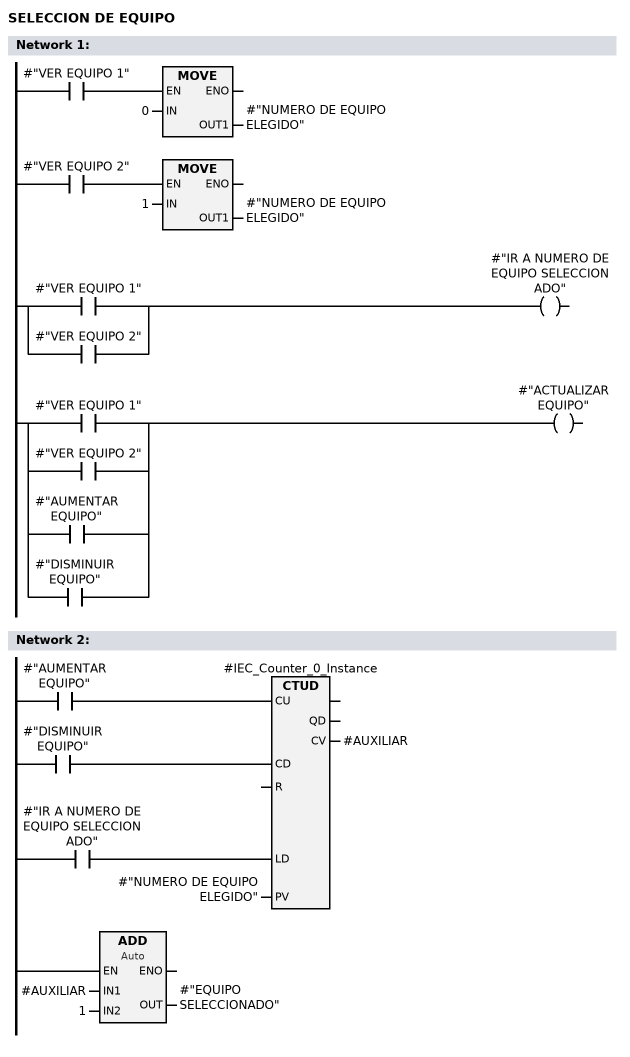
   RUNG wire#powerrail
      Contact( #"VER EQUIPO 1" )
      Move(in := 0, out1 => #"NUMERO DE EQUIPO ELEGIDO")
   END_RUNG
   RUNG wire#powerrail
      Contact( #"VER EQUIPO 2" )
      Move(in := 1, out1 => #"NUMERO DE EQUIPO ELEGIDO")
   END_RUNG
   RUNG wire#powerrail
      Contact( #"VER EQUIPO 1" )
      wire#w1
      Coil( #"IR A NUMERO DE EQUIPO SELECCIONADO" )
   END_RUNG
   RUNG wire#powerrail
      Contact( #"VER EQUIPO 2" )
   END_RUNG wire#w1
   RUNG wire#powerrail
      Contact( #"VER EQUIPO 1" )
      wire#w2
      Coil( #"ACTUALIZAR EQUIPO" )
   END_RUNG
   RUNG wire#powerrail
      Contact( #"VER EQUIPO 2" )
   END_RUNG wire#w2
   RUNG wire#powerrail
      Contact( #"AUMENTAR EQUIPO" )
   END_RUNG wire#w2
   RUNG wire#powerrail
      Contact( #"DISMINUIR EQUIPO" )
   END_RUNG wire#w2
   // the same network as SCL:
   IF #"VER EQUIPO 1" THEN #"NUMERO DE EQUIPO ELEGIDO" := 0; END_IF;
   IF #"VER EQUIPO 2" THEN #"NUMERO DE EQUIPO ELEGIDO" := 1; END_IF;
   #"IR A NUMERO DE EQUIPO SELECCIONADO" := #"VER EQUIPO 1" OR #"VER EQUIPO 2";
   #"ACTUALIZAR EQUIPO" := #"VER EQUIPO 1" OR #"VER EQUIPO 2" OR #"AUMENTAR EQUIPO" OR #"DISMINUIR EQUIPO";
END_REGION

REGION Network 2
   #IEC_Counter_0_Instance(CU := #"AUMENTAR EQUIPO",   // CTUD
                           CD := #"DISMINUIR EQUIPO",
                           LD := #"IR A NUMERO DE EQUIPO SELECCIONADO",
                           PV := #"NUMERO DE EQUIPO ELEGIDO",
                           CV => #AUXILIAR);
   #"EQUIPO SELECCIONADO" := #AUXILIAR + 1;
END_REGION
END_FUNCTION_BLOCK

FUNCTION_BLOCK "NIVEL DE AGUA"   // FB3, LAD
{ S7_Optimized_Access := 'TRUE' }
VERSION : 0.1
   VAR_INPUT
      "INPUT SENSOR" : Int;
      "CALIBRAR MAXIMO" : Bool;
      "CALIBRAR MINIMO" : Bool;
      "LARGO REGLA" : Int;
   END_VAR
   VAR_OUTPUT
      "ALTURA [mm]" : Int;
   END_VAR
   VAR
      IEC_Timer_0_Instance : TOF_TIME;
   END_VAR
   VAR RETAIN
      "AUXILIAR 1" : Real;
      TENSION : Real;
      "TENSION MAX REGLA" : Real;
      "TENSION MIN REGLA" : Real;
      "PENDIENTE RECTA" : Real;
      "ORDENADA AL ORIGEN" : Real;
      "AUXILIAR 2" : Real;
      "TENSION_LEER ALTURA" : Real;
      "ALTURA AUX [mm]" : Real;
      "COMPARADOR AUX" : Real;
   END_VAR
   VAR_TEMP   // added for the SCL form of the ladder/FBD networks
      _w1 : Bool;
      _w2 : Bool;
      _w3 : Bool;
      _w4 : Bool;
   END_VAR
BEGIN

REGION Network 1
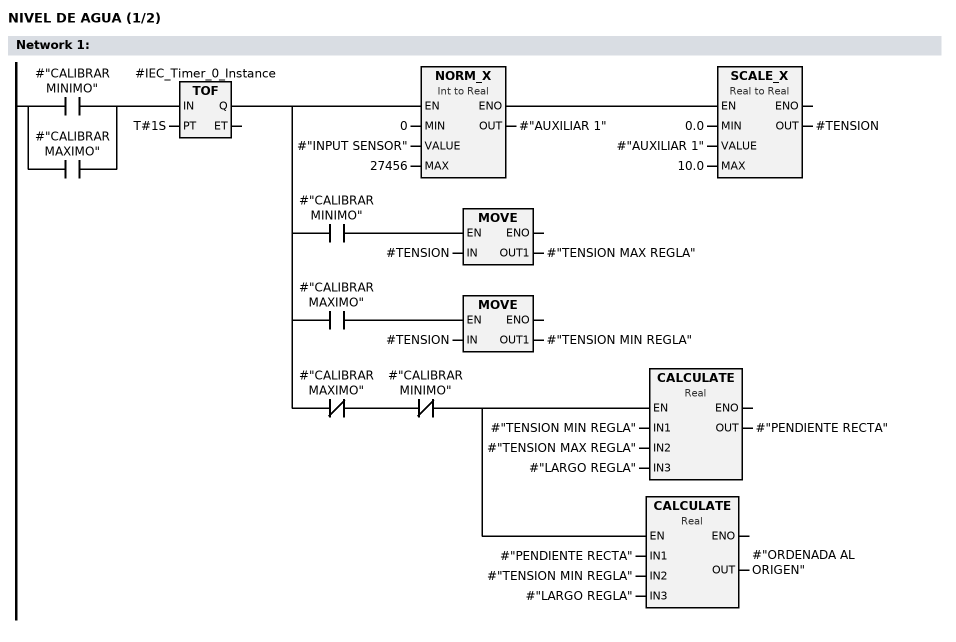
   #IEC_Timer_0_Instance(IN := #"CALIBRAR MINIMO" OR #"CALIBRAR MAXIMO", PT := T#1S);   // TOF
   IF #IEC_Timer_0_Instance.Q THEN
       #"AUXILIAR 1" := NORM_X(MIN := 0, VALUE := #"INPUT SENSOR", MAX := 27456);
       #TENSION := SCALE_X(MIN := 0.0, VALUE := #"AUXILIAR 1", MAX := 10.0);
   END_IF;
   IF #IEC_Timer_0_Instance.Q AND #"CALIBRAR MINIMO" THEN #"TENSION MAX REGLA" := #TENSION; END_IF;
   IF #IEC_Timer_0_Instance.Q AND #"CALIBRAR MAXIMO" THEN #"TENSION MIN REGLA" := #TENSION; END_IF;
   IF #IEC_Timer_0_Instance.Q AND NOT #"CALIBRAR MAXIMO" AND NOT #"CALIBRAR MINIMO" THEN
       #"PENDIENTE RECTA" := -#"LARGO REGLA"/(#"TENSION MAX REGLA"-#"TENSION MIN REGLA");
       #"ORDENADA AL ORIGEN" := #"LARGO REGLA"-#"TENSION MIN REGLA"*#"PENDIENTE RECTA";
   END_IF;
END_REGION

REGION Network 2: LEER ALTURA
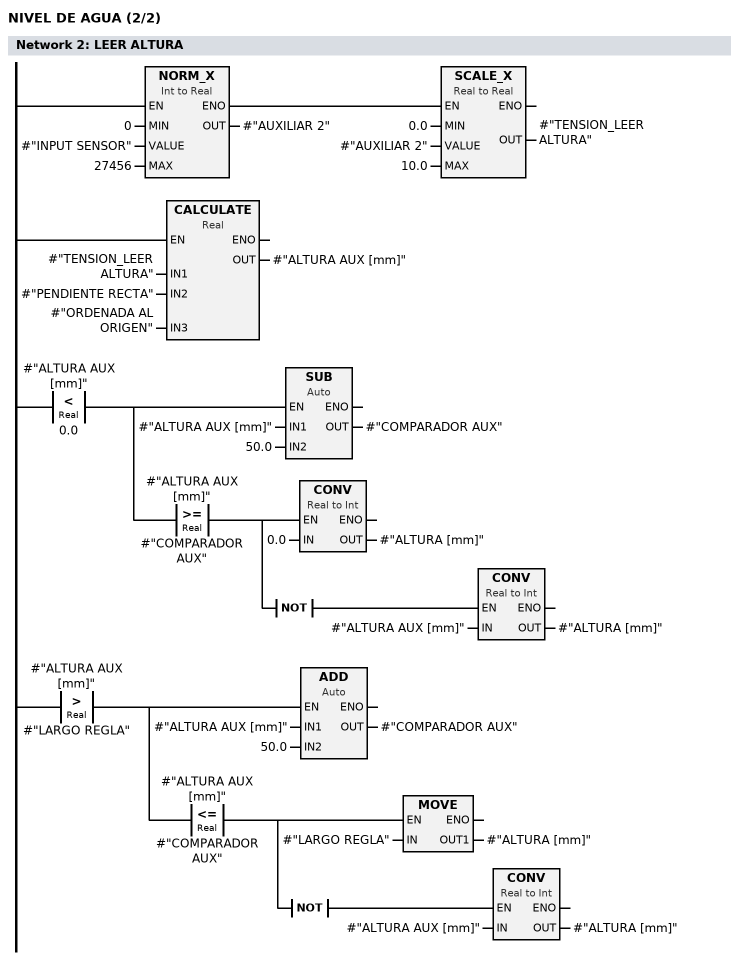
   RUNG wire#powerrail
      { S7_Templates := "[SrcType := Int, DestType := Real]" } Normalize(min := 0, value := #"INPUT SENSOR", max := 27456, out => #"AUXILIAR 2")
      { S7_Templates := "[SrcType := Real, DestType := Real]" } Scale(min := 0.0, value := #"AUXILIAR 2", max := 10.0, out => #"TENSION_LEER ALTURA")
   END_RUNG
   RUNG wire#powerrail
      { S7_Templates := "SrcType := Real"; S7_Expression := "IN1*IN2+IN3" } Calculate(in1 := #"TENSION_LEER ALTURA", in2 := #"PENDIENTE RECTA", in3 := #"ORDENADA AL ORIGEN", out => #"ALTURA AUX [mm]")
   END_RUNG
   RUNG wire#powerrail
      { S7_Templates := "SrcType := Real" } LT_Contact(in1 := #"ALTURA AUX [mm]", in2 := 0.0)
      wire#w1
      Sub(in1 := #"ALTURA AUX [mm]", in2 := 50.0, out => #"COMPARADOR AUX")
   END_RUNG
   RUNG wire#w1
      { S7_Templates := "SrcType := Real" } GE_Contact(in1 := #"ALTURA AUX [mm]", in2 := #"COMPARADOR AUX")
      wire#w2
      { S7_Templates := "[SrcType := Real, DestType := Int]" } Convert(in := 0.0, out => #"ALTURA [mm]")
   END_RUNG
   RUNG wire#w2
      Not()
      { S7_Templates := "[SrcType := Real, DestType := Int]" } Convert(in := #"ALTURA AUX [mm]", out => #"ALTURA [mm]")
   END_RUNG
   RUNG wire#powerrail
      { S7_Templates := "SrcType := Real" } GT_Contact(in1 := #"ALTURA AUX [mm]", in2 := #"LARGO REGLA")
      wire#w3
      Add(in1 := #"ALTURA AUX [mm]", in2 := 50.0, out => #"COMPARADOR AUX")
   END_RUNG
   RUNG wire#w3
      { S7_Templates := "SrcType := Real" } LE_Contact(in1 := #"ALTURA AUX [mm]", in2 := #"COMPARADOR AUX")
      wire#w4
      Move(in := #"LARGO REGLA", out1 => #"ALTURA [mm]")
   END_RUNG
   RUNG wire#w4
      Not()
      { S7_Templates := "[SrcType := Real, DestType := Int]" } Convert(in := #"ALTURA AUX [mm]", out => #"ALTURA [mm]")
   END_RUNG
   // the same network as SCL:
   #"AUXILIAR 2" := NORM_X(MIN := 0, VALUE := #"INPUT SENSOR", MAX := 27456);
   #"TENSION_LEER ALTURA" := SCALE_X(MIN := 0.0, VALUE := #"AUXILIAR 2", MAX := 10.0);
   #"ALTURA AUX [mm]" := #"TENSION_LEER ALTURA"*#"PENDIENTE RECTA"+#"ORDENADA AL ORIGEN";
   #_w1 := #"ALTURA AUX [mm]" < 0.0;
   IF #_w1 THEN #"COMPARADOR AUX" := #"ALTURA AUX [mm]" - 50.0; END_IF;
   #_w2 := #_w1 AND (#"ALTURA AUX [mm]" >= #"COMPARADOR AUX");
   IF #_w2 THEN #"ALTURA [mm]" := REAL_TO_INT(0.0); END_IF;
   IF NOT #_w2 THEN #"ALTURA [mm]" := REAL_TO_INT(#"ALTURA AUX [mm]"); END_IF;
   #_w3 := #"ALTURA AUX [mm]" > #"LARGO REGLA";
   IF #_w3 THEN #"COMPARADOR AUX" := #"ALTURA AUX [mm]" + 50.0; END_IF;
   #_w4 := #_w3 AND (#"ALTURA AUX [mm]" <= #"COMPARADOR AUX");
   IF #_w4 THEN #"ALTURA [mm]" := #"LARGO REGLA"; END_IF;
   IF NOT #_w4 THEN #"ALTURA [mm]" := REAL_TO_INT(#"ALTURA AUX [mm]"); END_IF;
END_REGION
END_FUNCTION_BLOCK

FUNCTION_BLOCK "FUNCION EQUIPO"   // FB4, LAD
{ S7_Optimized_Access := 'TRUE' }
VERSION : 0.1
   VAR_INPUT
      "PARAMETROS FUNCIONAMIENTO" : Array[1..4] of Struct   // Lo traslado a cada equipo desde HMI carga
         "CANTIDAD DE TORRES" : Int;
         "NIVEL MINIMO" : Array[1..3] of Int;   // El arreglo es porque hay 3 torres
         "TIPO DE CORTE" : Bool;
         "TEMPERATURA CORTE" : Int;
         "TIEMPO CORTE" : Int;
         "NUMERO RECETA" : Int;
         "NOMBRE RECETA" : String;
         "ESTADO ACTUAL" : String;
         "TIEMPO TOTAL TRANSCURRIDO" : Int;
         "PASO ACTUAL" : Int;
      END_STRUCT;
      CONFIGURACIONES : Array[1..4] of Struct
         DELAY : Int;
         HISTERESIS : DInt;
         "TIEMPO MAXIMO CICLO" : Int;
         "NIVEL CRITICO" : Int;
         "NIVEL PO" : Array[1..3] of Int;
         "NIVEL OP" : Int;
         VENTANA : Int;
      END_STRUCT;
      "RECETA  EQUIPOS" : Array[1..4] of Struct   // Se guarda la receta elegida en cada equipo
         PASOS : Int;
         "TEMP AGUA" : Array[1..4] of Int;
         "TEMP PRODUCTO" : Array[1..4] of Int;
         "TIEMPO CORTE" : Array[1..4] of Int;
         "TIPO CORTE" : Array[1..4] of Bool;
         NOMBRE : String;
         "TIEMPO CORTE ENFRIADO" : Int;
         "TEMP CORTE ENFRIADO" : Int;
         "TIPO CORTE ENFRIADO" : Bool;
      END_STRUCT;
      "NUMERO RECETA CARGADA" : Array[1..4] of Int;
      TEMPERATURAS : Array[1..4] of Struct
         "TEMPERATURA AGUA" : Real;
         "TEMPERATURA INGRESO" : Real;
         "TEMPERATURA PRODUCTO" : Real;
         "TEMPERATURA AGUA SC" : Real;
         "TEMPERATURA INGRESO SC" : Real;
         "TEMPERATURA PRODUCTO SC" : Real;
      END_STRUCT;
      NIVEL : Array[1..4] of Int;
      "SEÑALES ENTRADAS" : Struct
         "GUARDAMOTOR BI" : Array[1..4] of Bool;
         "GUARDAMOTOR BE" : Array[1..4] of Bool;
         "NIVEL BAJO CHILLER" : Array[1..4] of Bool;
         "NIVEL OK CHILLER" : Array[1..4] of Bool;
         "NIVEL REBALSE CHILLER" : Array[1..4] of Bool;
         "FALLA CHILLER" : Array[1..4] of Bool;
      END_STRUCT;
      "EQUIPO SELECCIONADO" : Int;
      "SCAN EQUIPOS" : Int;
      REARME : Bool;
      "INICIAR PRE OPERATIVO" : Bool;
      "INICIAR OPERATIVO" : Bool;
      PAUSA : Bool;
      CONTINUAR : Bool;
      CANCELAR : Bool;
      "PULSADOR EMERGENCIA" : Bool;
      "OK FIN CICLO" : Bool;
      "OK CANCELAR" : Bool;
   END_VAR
   VAR_OUTPUT
      ESTADO : Struct
         EQUIPOS : Array[1..4] of String;
         CHILLER : Array[1..4] of String;
      END_STRUCT;
      ACTUADORES : Array[1..4] of Struct
         "BALIZA VERDE" : Bool;
         "BALIZA ROJA" : Bool;
         BUZZER : Bool;
         "BOMBA RECIRCULACION" : Bool;
         "BOMBA EGRESO" : Bool;
         "BOMBA INGRESO" : Bool;
         "VAPOR SERPENTINA" : Bool;
         "VAPOR VIVO" : Bool;
         "VALVULA CARGA DE AGUA" : Bool;
         "TOMA FILTRO" : Bool;
         "INGRESO DE AGUA" : Bool;
         "EGRESO DE AGUA" : Bool;
         "NIVEL REBALSE CHILLER" : Bool;
         "NIVEL OPTIMO CHILLER" : Bool;
         "NIVEL BAJO CHILLER" : Bool;
      END_STRUCT;
      "SALIDA HISTERESIS MINIMA" : Array[1..4] of Int;
      "SALIDA HISTERESIS MAXIMA" : Array[1..4] of Int;
      "TIEMPOS TRANSCURRIDOS" : Array[1..4] of DInt;
   END_VAR
   VAR
      "NUMERO EQUIPO" : Int;
      "INICIAR CICLO PO" : Array[1..4] of Bool;
      "INICIAR CICLO OP" : Array[1..4] of Bool;
      "CICLO CANCELADO" : Array[1..4] of Bool;
      "PAUSAR CICLO" : Array[1..4] of Bool;
      "CONTINUAR CICLO" : Array[1..4] of Bool;
      "TIPO DE EQUIPO" : Array[1..4] of Bool;
      "PO POR TEMPERATURA" : Array[1..4] of Bool;
      "PO POR TIEMPO" : Array[1..4] of Bool;
      "TEMPERATURA PO ALCANZADA" : Array[1..4] of Bool;
      "PO EQUIPO 3" : TON_TIME;
      "PO EQUIPO 4" : TON_TIME;
      "PO EQUIPO 1" : TONR_TIME;
      "PO EQUIPO 2" : TONR_TIME;
      "TIEMPO CORTE EQUIPO" : Array[1..4] of DInt;
      "TIEMPO PO ALCANZADO" : Array[1..4] of Bool;
      "NIVEL PO A ALCANZAR" : Array[1..4] of Int;
      "NIVEL DE AGUA PO ALCANZADO" : Array[1..4] of Bool;
      "NIVEL DE AGUA OP ALCANZADO" : Array[1..4] of Bool;
      "CARGANDO AGUA" : Array[1..4] of Bool;
      "NIVEL OP A ALCANZAR" : Array[1..4] of Int;
   END_VAR
   VAR RETAIN
      "CONTADOR PASOS EQUIPO 1" : CTU_INT;
      "CONTADOR DE PASOS EQUIPO 2" : CTU_INT;
   END_VAR
   VAR
      "PASO ACTUAL" : Array[1..4] of Int;
      "HISTERESIS MAXIMA" : Array[1..4] of Int;
      "HISTERESIS MINIMA" : Array[1..4] of Int;
      "TEMPERATURA PASO ALCANZADA" : Array[1..4] of Bool;
      "AUXILIAR 1" : Int;
      "AUXILIAR 2" : Int;
      "AUXILIAR 3" : Int;
      "AUXILIAR 4" : Int;
   END_VAR
   VAR RETAIN
      "CONTADOR DE PASOS EQUIPO 3" : CTU_INT;
      "CONTADOR DE PASOS EQUIPO 4" : CTU_INT;
   END_VAR
   VAR
      "TIEMPO PASO OP EQUIPO 1" : TON_TIME;
      "TIEMPO PASO OP EQUIPO 2" : TON_TIME;
      "TIEMPO PASO OP EQUIPO 3" : TON_TIME;
      "TIEMPO PASO OP EQUIPO 4" : TON_TIME;
      "TIEMPO CORTE OP" : Array[1..4] of DInt;
      "AUXILIAR 5" : DInt;
      "NIVEL ALTO" : Array[1..4] of Bool;
      "NIVEL OK" : Array[1..4] of Bool;
      "NIVEL BAJO" : Array[1..4] of Bool;
      "NIVEL MAXIMO DE AGUA" : Array[1..4] of Int;
      "NIVEL MINIMO DE AGUA" : Array[1..4] of Int;
      "NIVEL FUNCIONAMIENTO" : Array[1..4] of Int;
      IEC_Timer_0_Instance_4 : TON_TIME;
      IEC_Timer_0_Instance_5 : TOF_TIME;
      IEC_Timer_0_Instance_6 : TON_TIME;
      IEC_Timer_0_Instance_7 : TOF_TIME;
      IEC_Timer_0_Instance_8 : TON_TIME;
      IEC_Timer_0_Instance_9 : TOF_TIME;
      IEC_Timer_0_Instance_10 : TON_TIME;
      IEC_Timer_0_Instance_11 : TOF_TIME;
      "AUXILIAR VS" : Array[1..4] of Bool;
      "AUXILIAR BOMBA INGRESO" : Array[1..4] of Bool;
      "AUXILIAR BOMBA EGRESO" : Array[1..4] of Bool;
      "PREPARACION NIVEL CHILLER" : Array[1..4] of Bool;
      "SUMINISTRAR AGUA A CHILLER" : Array[1..4] of Bool;
      FALLA : Array[1..4] of Bool;
      "NIVEL CHILLER ALCANZADO" : Array[1..4] of Bool;
      "EN CICLO" : Array[1..4] of Bool;
      "CONTROL NIVEL CARGA DE CHILLER" : Array[1..4] of Bool;
      "TIEMPO PASO ALCANZADA" : Array[1..4] of Bool;
      "PASOS COMPLETADOS" : Array[1..4] of Bool;
      "NIVEL REBALSE" : Array[1..4] of Bool;
      "CICLO PO FINALIZADO" : Array[1..4] of Bool;
      "CICLO OP FINALIZADO" : Array[1..4] of Bool;
      "RESET FIN CICLO" : Array[1..4] of Bool;
      DELAY : Array[1..4] of DInt;
      IEC_Timer_0_Instance : TON_TIME;
      IEC_Timer_0_Instance_1 : TON_TIME;
   END_VAR
   VAR CONSTANT
      COCINA : String;
      "NIVEL COMIENZO CARGA A CHILLER" : Int := 400;
      "NIVEL CORTECARGA A CHILLER" : Int := 100;
      REBALSE : String := 'REBALSE';
      OK : String := 'OK';
      BAJO : String := 'BAJO';
      "PRE OPERATIVO" : String := 'PRE OPERATIVO';
      OPERATIVO : String := 'OPERATIVO';
      PAUSADO : String := 'PAUSADO';
      INACTIVO : String := 'INACTIVO';
      "FIN PRE OPERATIVO" : String := 'FIN PRE OPERATIVO';
      "FIN OPERATIVO" : String := 'FIN OPERATIVO';
   END_VAR
   VAR_TEMP   // added for the SCL form of the ladder/FBD networks
      _w1 : Bool;
      _w2 : Bool;
   END_VAR
   // // "PARAMETROS FUNCIONAMIENTO"[1] : Cada equipo con sus configuraciones en
   // // CONFIGURACIONES[1]."NIVEL PO"[1] : Nivel PO para 1 torre
   // // CONFIGURACIONES[1]."NIVEL PO"[2] : Nivel PO para 2 torres
   // // CONFIGURACIONES[1]."NIVEL PO"[3] : Nivel PO para 3 torres
BEGIN

REGION Network 1: TIPO DE EQUIPO
   // TIPO DE EQUIPO 
   // 0 - ENFRIADOR
   // 1 - COCINA
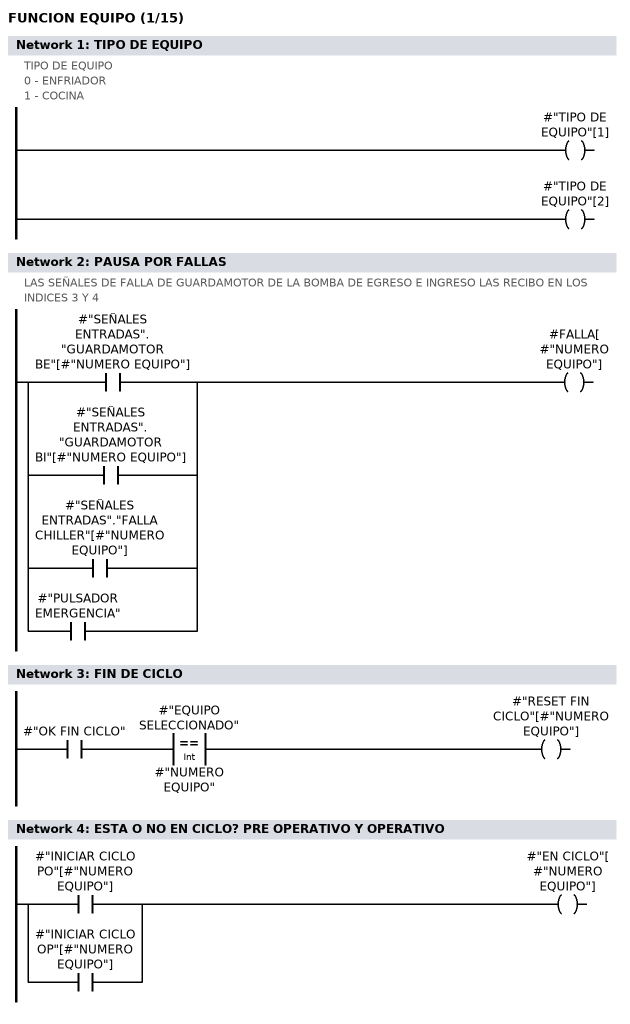
   RUNG wire#powerrail
      Coil( #"TIPO DE EQUIPO"[1] )
   END_RUNG
   RUNG wire#powerrail
      Coil( #"TIPO DE EQUIPO"[2] )
   END_RUNG
   // the same network as SCL:
   #"TIPO DE EQUIPO"[1] := TRUE;
   #"TIPO DE EQUIPO"[2] := TRUE;
END_REGION

REGION Network 2: PAUSA POR FALLAS
   // LAS SEÑALES DE FALLA DE GUARDAMOTOR DE LA BOMBA DE EGRESO E INGRESO LAS RECIBO EN LOS INDICES 3 Y 4
   RUNG wire#powerrail
      Contact( #"SEÑALES ENTRADAS"."GUARDAMOTOR BE"[#"NUMERO EQUIPO"] )
      wire#w1
      Coil( #FALLA[#"NUMERO EQUIPO"] )
   END_RUNG
   RUNG wire#powerrail
      Contact( #"SEÑALES ENTRADAS"."GUARDAMOTOR BI"[#"NUMERO EQUIPO"] )
   END_RUNG wire#w1
   RUNG wire#powerrail
      Contact( #"SEÑALES ENTRADAS"."FALLA CHILLER"[#"NUMERO EQUIPO"] )
   END_RUNG wire#w1
   RUNG wire#powerrail
      Contact( #"PULSADOR EMERGENCIA" )
   END_RUNG wire#w1
   // the same network as SCL:
   #FALLA[#"NUMERO EQUIPO"] := #"SEÑALES ENTRADAS"."GUARDAMOTOR BE"[#"NUMERO EQUIPO"] OR #"SEÑALES ENTRADAS"."GUARDAMOTOR BI"[#"NUMERO EQUIPO"] OR #"SEÑALES ENTRADAS"."FALLA CHILLER"[#"NUMERO EQUIPO"] OR #"PULSADOR EMERGENCIA";
END_REGION

REGION Network 3: FIN DE CICLO
   RUNG wire#powerrail
      Contact( #"OK FIN CICLO" )
      { S7_Templates := "SrcType := Int" } EQ_Contact(in1 := #"EQUIPO SELECCIONADO", in2 := #"NUMERO EQUIPO")
      Coil( #"RESET FIN CICLO"[#"NUMERO EQUIPO"] )
   END_RUNG
   // the same network as SCL:
   #"RESET FIN CICLO"[#"NUMERO EQUIPO"] := #"OK FIN CICLO" AND (#"EQUIPO SELECCIONADO" = #"NUMERO EQUIPO");
END_REGION

REGION Network 4: ESTA O NO EN CICLO? PRE OPERATIVO Y OPERATIVO
   RUNG wire#powerrail
      Contact( #"INICIAR CICLO PO"[#"NUMERO EQUIPO"] )
      wire#w1
      Coil( #"EN CICLO"[#"NUMERO EQUIPO"] )
   END_RUNG
   RUNG wire#powerrail
      Contact( #"INICIAR CICLO OP"[#"NUMERO EQUIPO"] )
   END_RUNG wire#w1
   // the same network as SCL:
   #"EN CICLO"[#"NUMERO EQUIPO"] := #"INICIAR CICLO PO"[#"NUMERO EQUIPO"] OR #"INICIAR CICLO OP"[#"NUMERO EQUIPO"];
END_REGION

REGION Network 5: CONTROL Y COMIENZOS DE CICLOS
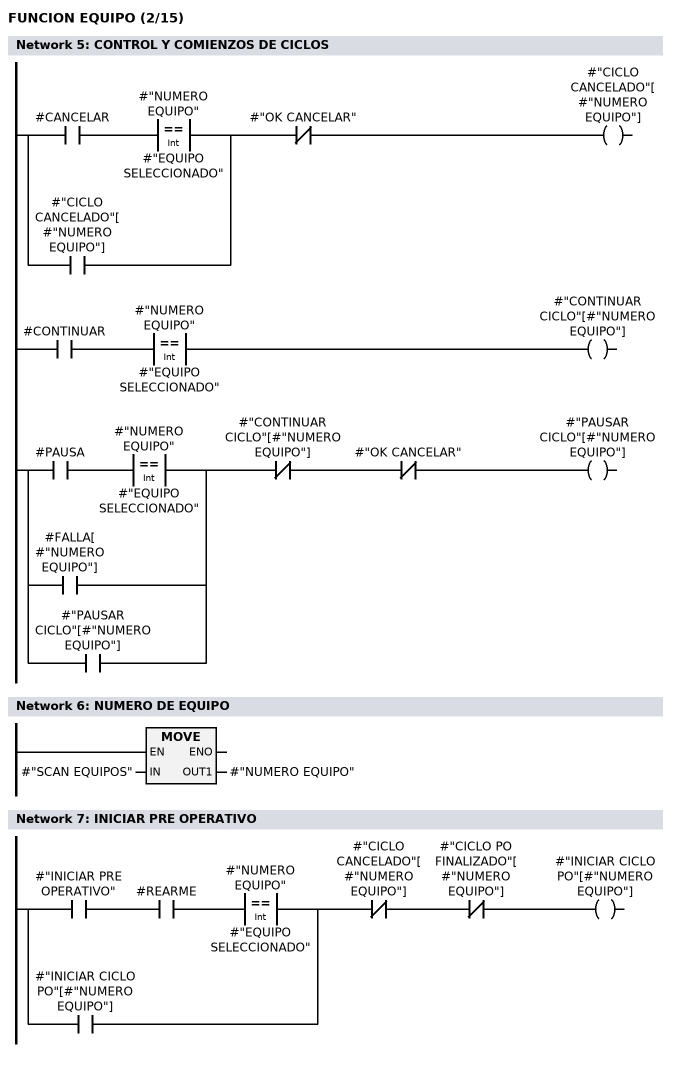
   RUNG wire#powerrail
      Contact( #CANCELAR )
      { S7_Templates := "SrcType := Int" } EQ_Contact(in1 := #"NUMERO EQUIPO", in2 := #"EQUIPO SELECCIONADO")
      wire#w1
      I_Contact( #"OK CANCELAR" )
      Coil( #"CICLO CANCELADO"[#"NUMERO EQUIPO"] )
   END_RUNG
   RUNG wire#powerrail
      Contact( #"CICLO CANCELADO"[#"NUMERO EQUIPO"] )
   END_RUNG wire#w1
   RUNG wire#powerrail
      Contact( #CONTINUAR )
      { S7_Templates := "SrcType := Int" } EQ_Contact(in1 := #"NUMERO EQUIPO", in2 := #"EQUIPO SELECCIONADO")
      Coil( #"CONTINUAR CICLO"[#"NUMERO EQUIPO"] )
   END_RUNG
   RUNG wire#powerrail
      Contact( #PAUSA )
      { S7_Templates := "SrcType := Int" } EQ_Contact(in1 := #"NUMERO EQUIPO", in2 := #"EQUIPO SELECCIONADO")
      wire#w2
      I_Contact( #"CONTINUAR CICLO"[#"NUMERO EQUIPO"] )
      I_Contact( #"OK CANCELAR" )
      Coil( #"PAUSAR CICLO"[#"NUMERO EQUIPO"] )
   END_RUNG
   RUNG wire#powerrail
      Contact( #FALLA[#"NUMERO EQUIPO"] )
   END_RUNG wire#w2
   RUNG wire#powerrail
      Contact( #"PAUSAR CICLO"[#"NUMERO EQUIPO"] )
   END_RUNG wire#w2
   // the same network as SCL:
   #"CICLO CANCELADO"[#"NUMERO EQUIPO"] := ((#CANCELAR AND (#"NUMERO EQUIPO" = #"EQUIPO SELECCIONADO")) OR #"CICLO CANCELADO"[#"NUMERO EQUIPO"]) AND NOT #"OK CANCELAR";
   #"CONTINUAR CICLO"[#"NUMERO EQUIPO"] := #CONTINUAR AND (#"NUMERO EQUIPO" = #"EQUIPO SELECCIONADO");
   #"PAUSAR CICLO"[#"NUMERO EQUIPO"] := ((#PAUSA AND (#"NUMERO EQUIPO" = #"EQUIPO SELECCIONADO")) OR #FALLA[#"NUMERO EQUIPO"] OR #"PAUSAR CICLO"[#"NUMERO EQUIPO"]) AND NOT #"CONTINUAR CICLO"[#"NUMERO EQUIPO"] AND NOT #"OK CANCELAR";
END_REGION

REGION Network 6: NUMERO DE EQUIPO
   RUNG wire#powerrail
      Move(in := #"SCAN EQUIPOS", out1 => #"NUMERO EQUIPO")
   END_RUNG
   // the same network as SCL:
   #"NUMERO EQUIPO" := #"SCAN EQUIPOS";
END_REGION

REGION Network 7: INICIAR PRE OPERATIVO
   RUNG wire#powerrail
      Contact( #"INICIAR PRE OPERATIVO" )
      Contact( #REARME )
      { S7_Templates := "SrcType := Int" } EQ_Contact(in1 := #"NUMERO EQUIPO", in2 := #"EQUIPO SELECCIONADO")
      wire#w1
      I_Contact( #"CICLO CANCELADO"[#"NUMERO EQUIPO"] )
      I_Contact( #"CICLO PO FINALIZADO"[#"NUMERO EQUIPO"] )
      Coil( #"INICIAR CICLO PO"[#"NUMERO EQUIPO"] )
   END_RUNG
   RUNG wire#powerrail
      Contact( #"INICIAR CICLO PO"[#"NUMERO EQUIPO"] )
   END_RUNG wire#w1
   // the same network as SCL:
   #"INICIAR CICLO PO"[#"NUMERO EQUIPO"] := ((#"INICIAR PRE OPERATIVO" AND #REARME AND (#"NUMERO EQUIPO" = #"EQUIPO SELECCIONADO")) OR #"INICIAR CICLO PO"[#"NUMERO EQUIPO"]) AND NOT #"CICLO CANCELADO"[#"NUMERO EQUIPO"] AND NOT #"CICLO PO FINALIZADO"[#"NUMERO EQUIPO"];
END_REGION

REGION Network 8: FUNCION LLENAR CHILLER **************
   // NI BIEN ARRANCO EL CICLO, ME FIJO SI ESTA EN NIVEL OPTIMO
   // 
   // 
   // CON EL TIPO DE EQUIPO CLASIFICO Y SOLAMENTE LO HAGO PARA LOS ENFRIADORES EN LOS INDICES 3 Y 4
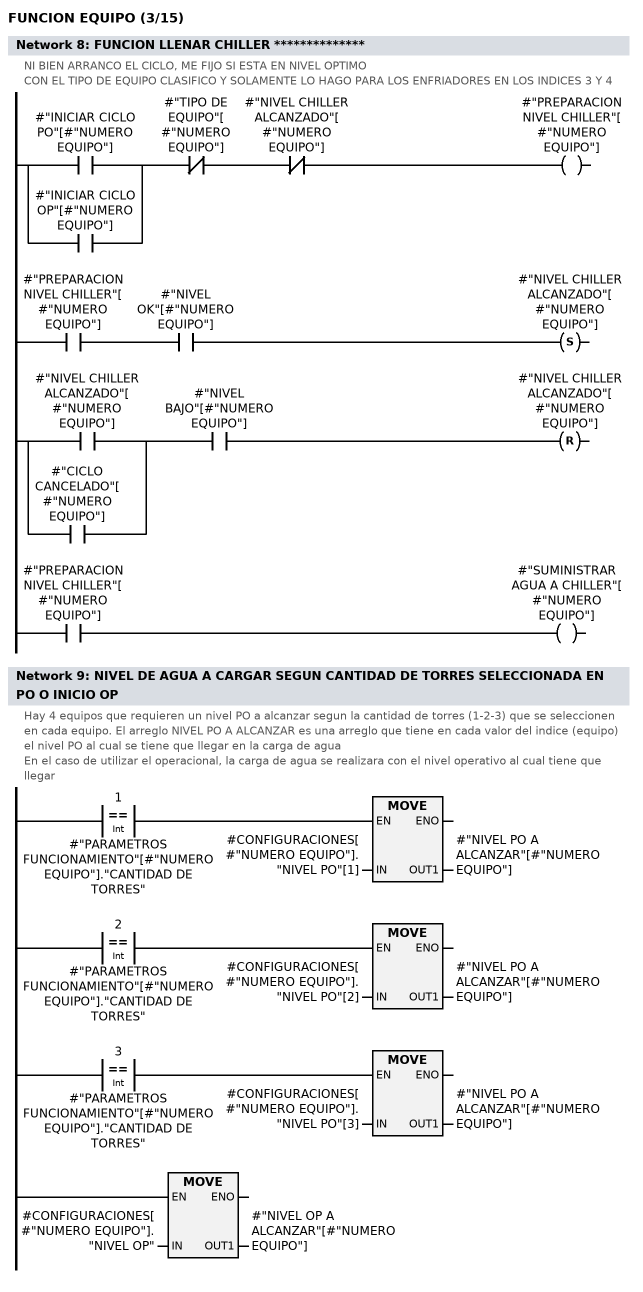
   RUNG wire#powerrail
      Contact( #"INICIAR CICLO PO"[#"NUMERO EQUIPO"] )
      wire#w1
      I_Contact( #"TIPO DE EQUIPO"[#"NUMERO EQUIPO"] )
      I_Contact( #"NIVEL CHILLER ALCANZADO"[#"NUMERO EQUIPO"] )
      Coil( #"PREPARACION NIVEL CHILLER"[#"NUMERO EQUIPO"] )
   END_RUNG
   RUNG wire#powerrail
      Contact( #"INICIAR CICLO OP"[#"NUMERO EQUIPO"] )
   END_RUNG wire#w1
   RUNG wire#powerrail
      Contact( #"PREPARACION NIVEL CHILLER"[#"NUMERO EQUIPO"] )
      Contact( #"NIVEL OK"[#"NUMERO EQUIPO"] )
      S_Coil( #"NIVEL CHILLER ALCANZADO"[#"NUMERO EQUIPO"] )
   END_RUNG
   RUNG wire#powerrail
      Contact( #"NIVEL CHILLER ALCANZADO"[#"NUMERO EQUIPO"] )
      wire#w2
      Contact( #"NIVEL BAJO"[#"NUMERO EQUIPO"] )
      R_Coil( #"NIVEL CHILLER ALCANZADO"[#"NUMERO EQUIPO"] )
   END_RUNG
   RUNG wire#powerrail
      Contact( #"CICLO CANCELADO"[#"NUMERO EQUIPO"] )
   END_RUNG wire#w2
   RUNG wire#powerrail
      Contact( #"PREPARACION NIVEL CHILLER"[#"NUMERO EQUIPO"] )
      Coil( #"SUMINISTRAR AGUA A CHILLER"[#"NUMERO EQUIPO"] )
   END_RUNG
   // the same network as SCL:
   #"PREPARACION NIVEL CHILLER"[#"NUMERO EQUIPO"] := (#"INICIAR CICLO PO"[#"NUMERO EQUIPO"] OR #"INICIAR CICLO OP"[#"NUMERO EQUIPO"]) AND NOT #"TIPO DE EQUIPO"[#"NUMERO EQUIPO"] AND NOT #"NIVEL CHILLER ALCANZADO"[#"NUMERO EQUIPO"];
   IF #"PREPARACION NIVEL CHILLER"[#"NUMERO EQUIPO"] AND #"NIVEL OK"[#"NUMERO EQUIPO"] THEN
       #"NIVEL CHILLER ALCANZADO"[#"NUMERO EQUIPO"] := TRUE;
   END_IF;
   IF (#"NIVEL CHILLER ALCANZADO"[#"NUMERO EQUIPO"] OR #"CICLO CANCELADO"[#"NUMERO EQUIPO"]) AND #"NIVEL BAJO"[#"NUMERO EQUIPO"] THEN
       #"NIVEL CHILLER ALCANZADO"[#"NUMERO EQUIPO"] := FALSE;
   END_IF;
   #"SUMINISTRAR AGUA A CHILLER"[#"NUMERO EQUIPO"] := #"PREPARACION NIVEL CHILLER"[#"NUMERO EQUIPO"];
END_REGION

REGION Network 9: NIVEL DE AGUA A CARGAR SEGUN CANTIDAD DE TORRES SELECCIONADA EN PO O INICIO OP
   // Hay 4 equipos que requieren un nivel PO a alcanzar segun la cantidad de torres (1-2-3) que se seleccionen en cada equipo. El arreglo NIVEL PO A ALCANZAR es una arreglo que tiene en cada valor del indice (equipo) el nivel PO al cual se tiene que llegar en la carga de agua
   // En el caso de utilizar el operacional, la carga de agua se realizara con el nivel operativo al cual tiene que llegar
   RUNG wire#powerrail
      { S7_Templates := "SrcType := Int" } EQ_Contact(in1 := 1, in2 := #"PARAMETROS FUNCIONAMIENTO"[#"NUMERO EQUIPO"]."CANTIDAD DE TORRES")
      Move(in := #CONFIGURACIONES[#"NUMERO EQUIPO"]."NIVEL PO"[1], out1 => #"NIVEL PO A ALCANZAR"[#"NUMERO EQUIPO"])
   END_RUNG
   RUNG wire#powerrail
      { S7_Templates := "SrcType := Int" } EQ_Contact(in1 := 2, in2 := #"PARAMETROS FUNCIONAMIENTO"[#"NUMERO EQUIPO"]."CANTIDAD DE TORRES")
      Move(in := #CONFIGURACIONES[#"NUMERO EQUIPO"]."NIVEL PO"[2], out1 => #"NIVEL PO A ALCANZAR"[#"NUMERO EQUIPO"])
   END_RUNG
   RUNG wire#powerrail
      { S7_Templates := "SrcType := Int" } EQ_Contact(in1 := 3, in2 := #"PARAMETROS FUNCIONAMIENTO"[#"NUMERO EQUIPO"]."CANTIDAD DE TORRES")
      Move(in := #CONFIGURACIONES[#"NUMERO EQUIPO"]."NIVEL PO"[3], out1 => #"NIVEL PO A ALCANZAR"[#"NUMERO EQUIPO"])
   END_RUNG
   RUNG wire#powerrail
      Move(in := #CONFIGURACIONES[#"NUMERO EQUIPO"]."NIVEL OP", out1 => #"NIVEL OP A ALCANZAR"[#"NUMERO EQUIPO"])
   END_RUNG
   // the same network as SCL:
   IF 1 = #"PARAMETROS FUNCIONAMIENTO"[#"NUMERO EQUIPO"]."CANTIDAD DE TORRES" THEN
       #"NIVEL PO A ALCANZAR"[#"NUMERO EQUIPO"] := #CONFIGURACIONES[#"NUMERO EQUIPO"]."NIVEL PO"[1];
   END_IF;
   IF 2 = #"PARAMETROS FUNCIONAMIENTO"[#"NUMERO EQUIPO"]."CANTIDAD DE TORRES" THEN
       #"NIVEL PO A ALCANZAR"[#"NUMERO EQUIPO"] := #CONFIGURACIONES[#"NUMERO EQUIPO"]."NIVEL PO"[2];
   END_IF;
   IF 3 = #"PARAMETROS FUNCIONAMIENTO"[#"NUMERO EQUIPO"]."CANTIDAD DE TORRES" THEN
       #"NIVEL PO A ALCANZAR"[#"NUMERO EQUIPO"] := #CONFIGURACIONES[#"NUMERO EQUIPO"]."NIVEL PO"[3];
   END_IF;
   #"NIVEL OP A ALCANZAR"[#"NUMERO EQUIPO"] := #CONFIGURACIONES[#"NUMERO EQUIPO"]."NIVEL OP";
END_REGION

REGION Network 10: CARGA DE AGUA ************* VER FUNCION
   // TENGO QUE TOCAR EL NIVEL DE AGUA ALCANZADO POR EL EQUIPO
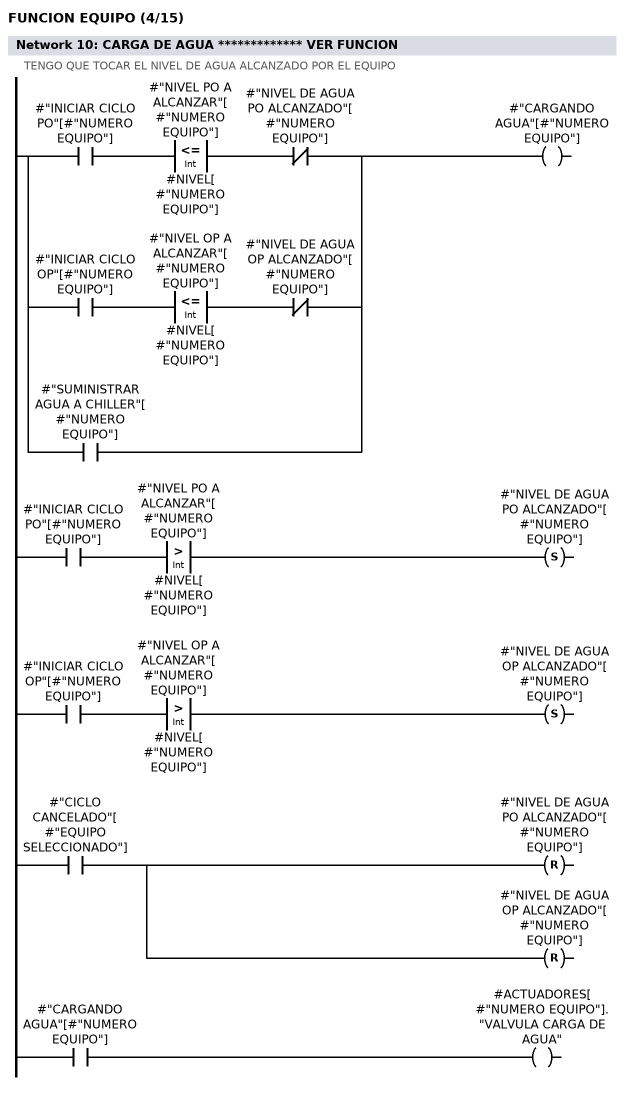
   RUNG wire#powerrail
      Contact( #"INICIAR CICLO PO"[#"NUMERO EQUIPO"] )
      { S7_Templates := "SrcType := Int" } LE_Contact(in1 := #"NIVEL PO A ALCANZAR"[#"NUMERO EQUIPO"], in2 := #NIVEL[#"NUMERO EQUIPO"])
      I_Contact( #"NIVEL DE AGUA PO ALCANZADO"[#"NUMERO EQUIPO"] )
      wire#w1
      Coil( #"CARGANDO AGUA"[#"NUMERO EQUIPO"] )
   END_RUNG
   RUNG wire#powerrail
      Contact( #"INICIAR CICLO OP"[#"NUMERO EQUIPO"] )
      { S7_Templates := "SrcType := Int" } LE_Contact(in1 := #"NIVEL OP A ALCANZAR"[#"NUMERO EQUIPO"], in2 := #NIVEL[#"NUMERO EQUIPO"])
      I_Contact( #"NIVEL DE AGUA OP ALCANZADO"[#"NUMERO EQUIPO"] )
   END_RUNG wire#w1
   RUNG wire#powerrail
      Contact( #"SUMINISTRAR AGUA A CHILLER"[#"NUMERO EQUIPO"] )
   END_RUNG wire#w1
   RUNG wire#powerrail
      Contact( #"INICIAR CICLO PO"[#"NUMERO EQUIPO"] )
      { S7_Templates := "SrcType := Int" } GT_Contact(in1 := #"NIVEL PO A ALCANZAR"[#"NUMERO EQUIPO"], in2 := #NIVEL[#"NUMERO EQUIPO"])
      S_Coil( #"NIVEL DE AGUA PO ALCANZADO"[#"NUMERO EQUIPO"] )
   END_RUNG
   RUNG wire#powerrail
      Contact( #"INICIAR CICLO OP"[#"NUMERO EQUIPO"] )
      { S7_Templates := "SrcType := Int" } GT_Contact(in1 := #"NIVEL OP A ALCANZAR"[#"NUMERO EQUIPO"], in2 := #NIVEL[#"NUMERO EQUIPO"])
      S_Coil( #"NIVEL DE AGUA OP ALCANZADO"[#"NUMERO EQUIPO"] )
   END_RUNG
   RUNG wire#powerrail
      Contact( #"CICLO CANCELADO"[#"EQUIPO SELECCIONADO"] )
      wire#w2
      R_Coil( #"NIVEL DE AGUA PO ALCANZADO"[#"NUMERO EQUIPO"] )
   END_RUNG
   RUNG wire#w2
      R_Coil( #"NIVEL DE AGUA OP ALCANZADO"[#"NUMERO EQUIPO"] )
   END_RUNG
   RUNG wire#powerrail
      Contact( #"CARGANDO AGUA"[#"NUMERO EQUIPO"] )
      Coil( #ACTUADORES[#"NUMERO EQUIPO"]."VALVULA CARGA DE AGUA" )
   END_RUNG
   // the same network as SCL:
   #"CARGANDO AGUA"[#"NUMERO EQUIPO"] := (#"INICIAR CICLO PO"[#"NUMERO EQUIPO"] AND (#"NIVEL PO A ALCANZAR"[#"NUMERO EQUIPO"] <= #NIVEL[#"NUMERO EQUIPO"]) AND NOT #"NIVEL DE AGUA PO ALCANZADO"[#"NUMERO EQUIPO"]) OR (#"INICIAR CICLO OP"[#"NUMERO EQUIPO"] AND (#"NIVEL OP A ALCANZAR"[#"NUMERO EQUIPO"] <= #NIVEL[#"NUMERO EQUIPO"]) AND NOT #"NIVEL DE AGUA OP ALCANZADO"[#"NUMERO EQUIPO"]) OR #"SUMINISTRAR AGUA A CHILLER"[#"NUMERO EQUIPO"];
   IF #"INICIAR CICLO PO"[#"NUMERO EQUIPO"] AND (#"NIVEL PO A ALCANZAR"[#"NUMERO EQUIPO"] > #NIVEL[#"NUMERO EQUIPO"]) THEN
       #"NIVEL DE AGUA PO ALCANZADO"[#"NUMERO EQUIPO"] := TRUE;
   END_IF;
   IF #"INICIAR CICLO OP"[#"NUMERO EQUIPO"] AND (#"NIVEL OP A ALCANZAR"[#"NUMERO EQUIPO"] > #NIVEL[#"NUMERO EQUIPO"]) THEN
       #"NIVEL DE AGUA OP ALCANZADO"[#"NUMERO EQUIPO"] := TRUE;
   END_IF;
   IF #"CICLO CANCELADO"[#"EQUIPO SELECCIONADO"] THEN
       #"NIVEL DE AGUA PO ALCANZADO"[#"NUMERO EQUIPO"] := FALSE;
       #"NIVEL DE AGUA OP ALCANZADO"[#"NUMERO EQUIPO"] := FALSE;
   END_IF;
   #ACTUADORES[#"NUMERO EQUIPO"]."VALVULA CARGA DE AGUA" := #"CARGANDO AGUA"[#"NUMERO EQUIPO"];
END_REGION

REGION Network 11: TIPO DE CORTE PRE OPERATIVO POR TEMPERATURA
   // BIT TIPO DE CORTE:
   // 
   // 0- TIEMPO
   // 1- TEMPERATURA
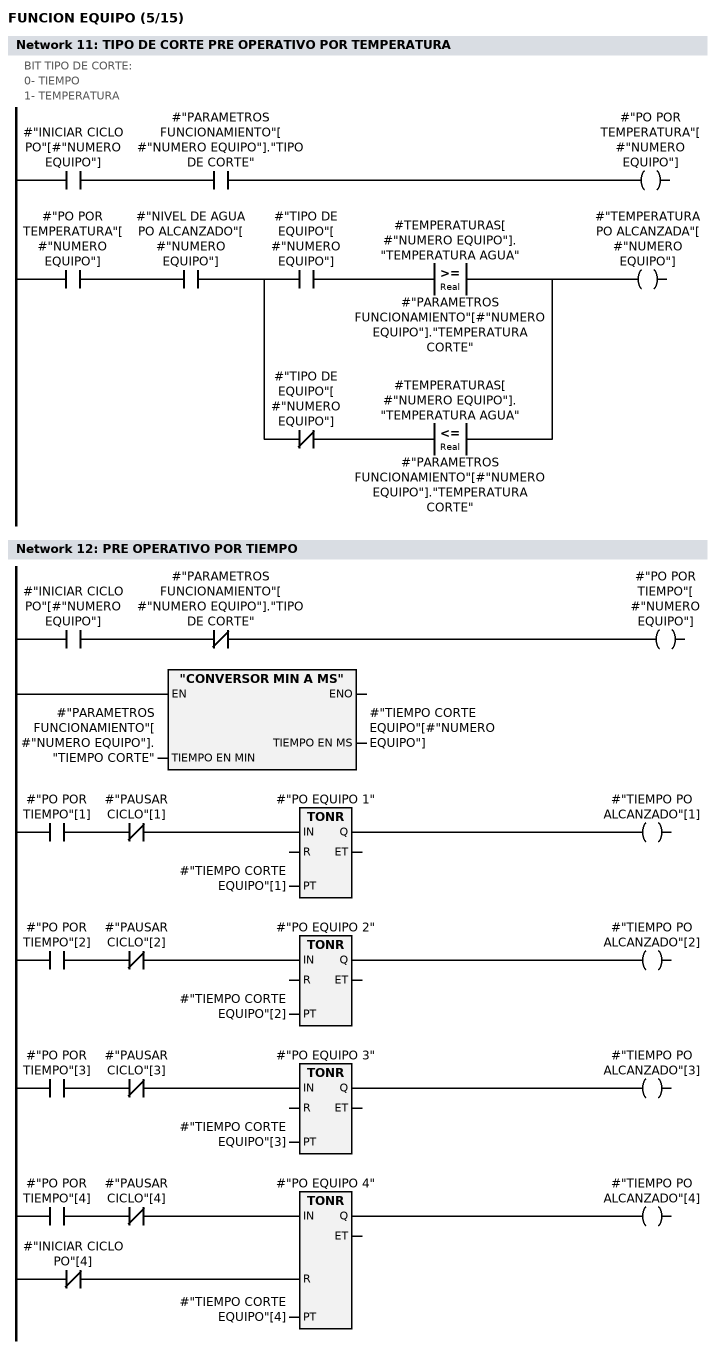
   RUNG wire#powerrail
      Contact( #"INICIAR CICLO PO"[#"NUMERO EQUIPO"] )
      Contact( #"PARAMETROS FUNCIONAMIENTO"[#"NUMERO EQUIPO"]."TIPO DE CORTE" )
      Coil( #"PO POR TEMPERATURA"[#"NUMERO EQUIPO"] )
   END_RUNG
   RUNG wire#powerrail
      Contact( #"PO POR TEMPERATURA"[#"NUMERO EQUIPO"] )
      Contact( #"NIVEL DE AGUA PO ALCANZADO"[#"NUMERO EQUIPO"] )
      wire#w1
      Contact( #"TIPO DE EQUIPO"[#"NUMERO EQUIPO"] )
      { S7_Templates := "SrcType := Real" } GE_Contact(in1 := #TEMPERATURAS[#"NUMERO EQUIPO"]."TEMPERATURA AGUA", in2 := #"PARAMETROS FUNCIONAMIENTO"[#"NUMERO EQUIPO"]."TEMPERATURA CORTE")
      wire#w2
      Coil( #"TEMPERATURA PO ALCANZADA"[#"NUMERO EQUIPO"] )
   END_RUNG
   RUNG wire#w1
      I_Contact( #"TIPO DE EQUIPO"[#"NUMERO EQUIPO"] )
      { S7_Templates := "SrcType := Real" } LE_Contact(in1 := #TEMPERATURAS[#"NUMERO EQUIPO"]."TEMPERATURA AGUA", in2 := #"PARAMETROS FUNCIONAMIENTO"[#"NUMERO EQUIPO"]."TEMPERATURA CORTE")
   END_RUNG wire#w2
   // the same network as SCL:
   #"PO POR TEMPERATURA"[#"NUMERO EQUIPO"] := #"INICIAR CICLO PO"[#"NUMERO EQUIPO"] AND #"PARAMETROS FUNCIONAMIENTO"[#"NUMERO EQUIPO"]."TIPO DE CORTE";
   #"TEMPERATURA PO ALCANZADA"[#"NUMERO EQUIPO"] := #"PO POR TEMPERATURA"[#"NUMERO EQUIPO"] AND #"NIVEL DE AGUA PO ALCANZADO"[#"NUMERO EQUIPO"] AND ((#"TIPO DE EQUIPO"[#"NUMERO EQUIPO"] AND (#TEMPERATURAS[#"NUMERO EQUIPO"]."TEMPERATURA AGUA" >= #"PARAMETROS FUNCIONAMIENTO"[#"NUMERO EQUIPO"]."TEMPERATURA CORTE")) OR (NOT #"TIPO DE EQUIPO"[#"NUMERO EQUIPO"] AND (#TEMPERATURAS[#"NUMERO EQUIPO"]."TEMPERATURA AGUA" <= #"PARAMETROS FUNCIONAMIENTO"[#"NUMERO EQUIPO"]."TEMPERATURA CORTE")));
END_REGION

REGION Network 12: PRE OPERATIVO POR TIEMPO
   #"PO POR TIEMPO"[#"NUMERO EQUIPO"] := #"INICIAR CICLO PO"[#"NUMERO EQUIPO"] AND NOT #"PARAMETROS FUNCIONAMIENTO"[#"NUMERO EQUIPO"]."TIPO DE CORTE";
   "CONVERSOR MIN A MS"("TIEMPO EN MIN" := #"PARAMETROS FUNCIONAMIENTO"[#"NUMERO EQUIPO"]."TIEMPO CORTE",
                        "TIEMPO EN MS" => #"TIEMPO CORTE EQUIPO"[#"NUMERO EQUIPO"]);
   #"PO EQUIPO 1"(IN := #"PO POR TIEMPO"[1] AND NOT #"PAUSAR CICLO"[1], PT := #"TIEMPO CORTE EQUIPO"[1]);   // TONR
   #"TIEMPO PO ALCANZADO"[1] := #"PO EQUIPO 1".Q;
   #"PO EQUIPO 2"(IN := #"PO POR TIEMPO"[2] AND NOT #"PAUSAR CICLO"[2], PT := #"TIEMPO CORTE EQUIPO"[2]);   // TONR
   #"TIEMPO PO ALCANZADO"[2] := #"PO EQUIPO 2".Q;
   #"PO EQUIPO 3"(IN := #"PO POR TIEMPO"[3] AND NOT #"PAUSAR CICLO"[3], PT := #"TIEMPO CORTE EQUIPO"[3]);   // TONR
   #"TIEMPO PO ALCANZADO"[3] := #"PO EQUIPO 3".Q;
   #"PO EQUIPO 4"(IN := #"PO POR TIEMPO"[4] AND NOT #"PAUSAR CICLO"[4],   // TONR
                  R := NOT #"INICIAR CICLO PO"[4],
                  PT := #"TIEMPO CORTE EQUIPO"[4]);
   #"TIEMPO PO ALCANZADO"[4] := #"PO EQUIPO 4".Q;
END_REGION

REGION Network 13: CICLO PO OPERATIVO FINALIZADO ***** FALTA HMI FIN CICLO
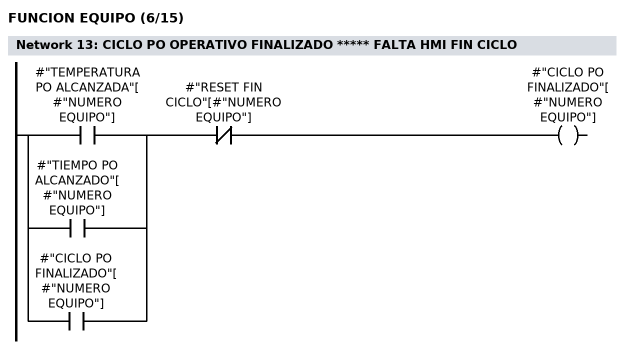
   RUNG wire#powerrail
      Contact( #"TEMPERATURA PO ALCANZADA"[#"NUMERO EQUIPO"] )
      wire#w1
      I_Contact( #"RESET FIN CICLO"[#"NUMERO EQUIPO"] )
      Coil( #"CICLO PO FINALIZADO"[#"NUMERO EQUIPO"] )
   END_RUNG
   RUNG wire#powerrail
      Contact( #"TIEMPO PO ALCANZADO"[#"NUMERO EQUIPO"] )
   END_RUNG wire#w1
   RUNG wire#powerrail
      Contact( #"CICLO PO FINALIZADO"[#"NUMERO EQUIPO"] )
   END_RUNG wire#w1
   // the same network as SCL:
   #"CICLO PO FINALIZADO"[#"NUMERO EQUIPO"] := (#"TEMPERATURA PO ALCANZADA"[#"NUMERO EQUIPO"] OR #"TIEMPO PO ALCANZADO"[#"NUMERO EQUIPO"] OR #"CICLO PO FINALIZADO"[#"NUMERO EQUIPO"]) AND NOT #"RESET FIN CICLO"[#"NUMERO EQUIPO"];
END_REGION

REGION Network 14: RECETAS CONTADOR DE PASOS
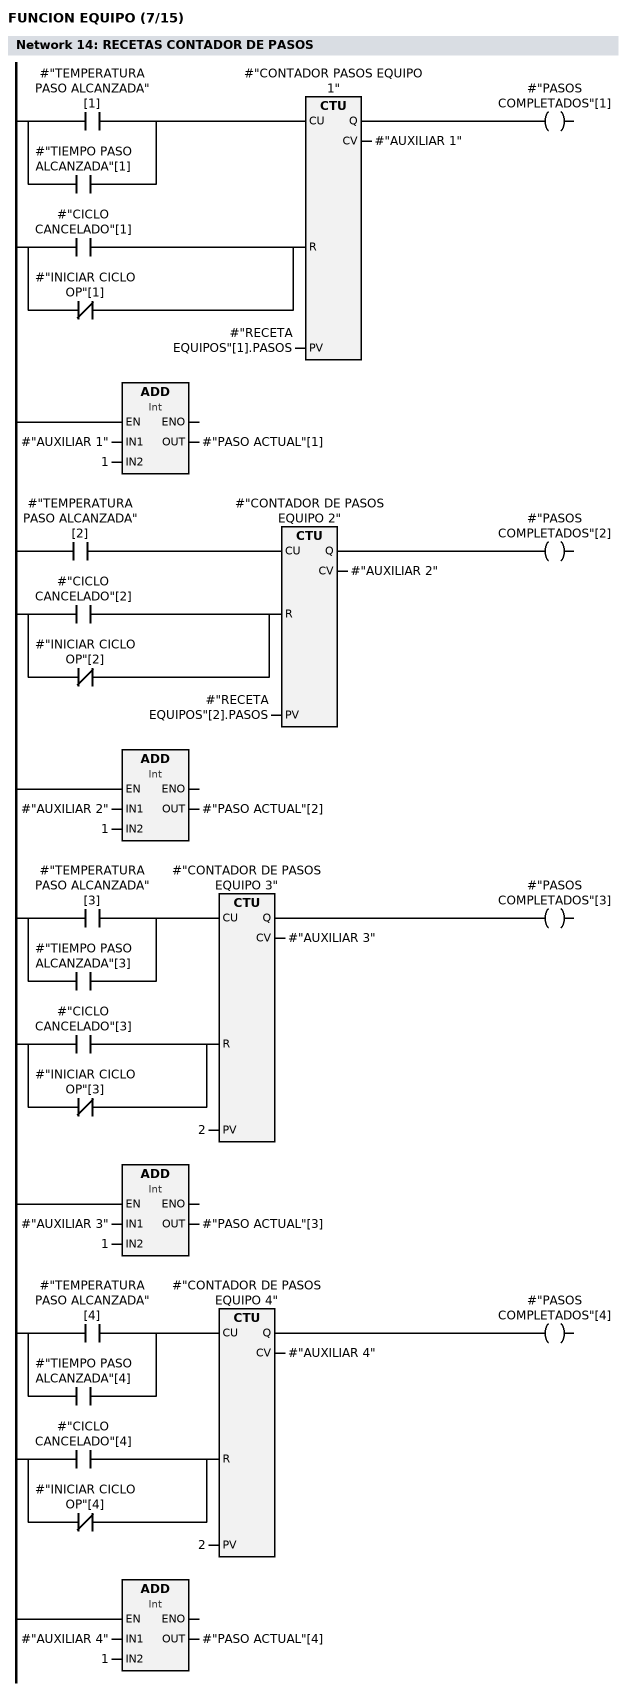
   #"CONTADOR PASOS EQUIPO 1"(CU := #"TEMPERATURA PASO ALCANZADA"[1] OR #"TIEMPO PASO ALCANZADA"[1],   // CTU
                           R := #"CICLO CANCELADO"[1] OR NOT #"INICIAR CICLO OP"[1],
                           PV := #"RECETA  EQUIPOS"[1].PASOS,
                           CV => #"AUXILIAR 1");
   #"PASOS COMPLETADOS"[1] := #"CONTADOR PASOS EQUIPO 1".Q;
   #"PASO ACTUAL"[1] := #"AUXILIAR 1" + 1;
   #"CONTADOR DE PASOS EQUIPO 2"(CU := #"TEMPERATURA PASO ALCANZADA"[2],   // CTU
                           R := #"CICLO CANCELADO"[2] OR NOT #"INICIAR CICLO OP"[2],
                           PV := #"RECETA  EQUIPOS"[2].PASOS,
                           CV => #"AUXILIAR 2");
   #"PASOS COMPLETADOS"[2] := #"CONTADOR DE PASOS EQUIPO 2".Q;
   #"PASO ACTUAL"[2] := #"AUXILIAR 2" + 1;
   #"CONTADOR DE PASOS EQUIPO 3"(CU := #"TEMPERATURA PASO ALCANZADA"[3] OR #"TIEMPO PASO ALCANZADA"[3],   // CTU
                           R := #"CICLO CANCELADO"[3] OR NOT #"INICIAR CICLO OP"[3],
                           PV := 2,
                           CV => #"AUXILIAR 3");
   #"PASOS COMPLETADOS"[3] := #"CONTADOR DE PASOS EQUIPO 3".Q;
   #"PASO ACTUAL"[3] := #"AUXILIAR 3" + 1;
   #"CONTADOR DE PASOS EQUIPO 4"(CU := #"TEMPERATURA PASO ALCANZADA"[4] OR #"TIEMPO PASO ALCANZADA"[4],   // CTU
                           R := #"CICLO CANCELADO"[4] OR NOT #"INICIAR CICLO OP"[4],
                           PV := 2,
                           CV => #"AUXILIAR 4");
   #"PASOS COMPLETADOS"[4] := #"CONTADOR DE PASOS EQUIPO 4".Q;
   #"PASO ACTUAL"[4] := #"AUXILIAR 4" + 1;
END_REGION

REGION Network 15: INICIO CICLO OP
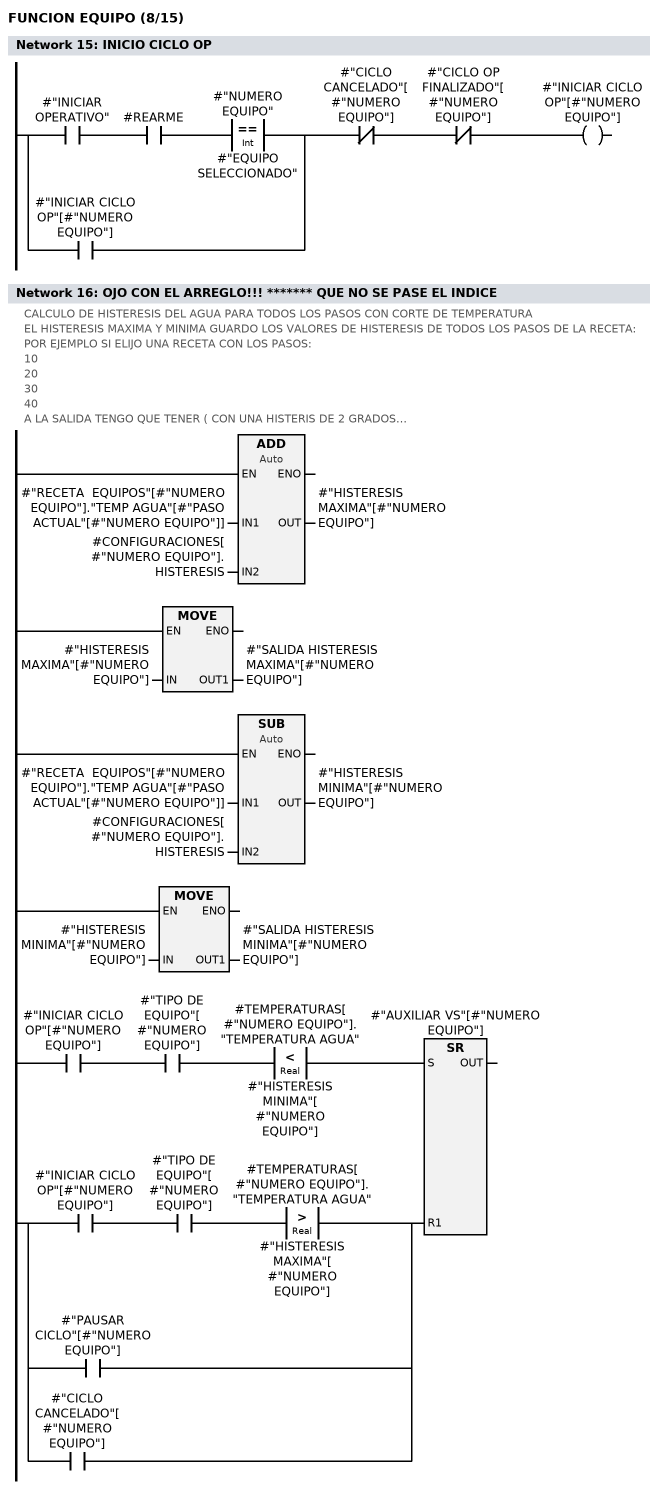
   RUNG wire#powerrail
      Contact( #"INICIAR OPERATIVO" )
      Contact( #REARME )
      { S7_Templates := "SrcType := Int" } EQ_Contact(in1 := #"NUMERO EQUIPO", in2 := #"EQUIPO SELECCIONADO")
      wire#w1
      I_Contact( #"CICLO CANCELADO"[#"NUMERO EQUIPO"] )
      I_Contact( #"CICLO OP FINALIZADO"[#"NUMERO EQUIPO"] )
      Coil( #"INICIAR CICLO OP"[#"NUMERO EQUIPO"] )
   END_RUNG
   RUNG wire#powerrail
      Contact( #"INICIAR CICLO OP"[#"NUMERO EQUIPO"] )
   END_RUNG wire#w1
   // the same network as SCL:
   #"INICIAR CICLO OP"[#"NUMERO EQUIPO"] := ((#"INICIAR OPERATIVO" AND #REARME AND (#"NUMERO EQUIPO" = #"EQUIPO SELECCIONADO")) OR #"INICIAR CICLO OP"[#"NUMERO EQUIPO"]) AND NOT #"CICLO CANCELADO"[#"NUMERO EQUIPO"] AND NOT #"CICLO OP FINALIZADO"[#"NUMERO EQUIPO"];
END_REGION

REGION Network 16: OJO CON EL ARREGLO!!! ******* QUE NO SE PASE EL INDICE
   // CALCULO DE HISTERESIS DEL AGUA PARA TODOS LOS PASOS CON CORTE DE TEMPERATURA
   // 
   // EL HISTERESIS MAXIMA Y MINIMA GUARDO LOS VALORES DE HISTERESIS DE TODOS LOS PASOS DE LA RECETA:
   // POR EJEMPLO SI ELIJO UNA RECETA CON LOS PASOS:
   // 10
   // 20
   // 30
   // 40
   // A LA SALIDA TENGO QUE TENER ( CON UNA HISTERIS DE 2 GRADOS)
   // 
   // HISTERESIS MINIMA:
   //  8
   // 18
   // 28
   // 38
   // 
   // HISTERESIS MAXIMA:
   // 12
   // 22
   // 32
   // 42
   // 
   // El auxiliar de vapor de serpentina lo utilizo porque el vapor de serpentina lo utilizo solamente en el estado operativo mientras que el vapor vivo lo utilizo en el pre operativo y operativo
   RUNG wire#powerrail
      Add(in1 := #"RECETA  EQUIPOS"[#"NUMERO EQUIPO"]."TEMP AGUA"[#"PASO ACTUAL"[#"NUMERO EQUIPO"]], in2 := #CONFIGURACIONES[#"NUMERO EQUIPO"].HISTERESIS, out => #"HISTERESIS MAXIMA"[#"NUMERO EQUIPO"])
   END_RUNG
   RUNG wire#powerrail
      Move(in := #"HISTERESIS MAXIMA"[#"NUMERO EQUIPO"], out1 => #"SALIDA HISTERESIS MAXIMA"[#"NUMERO EQUIPO"])
   END_RUNG
   RUNG wire#powerrail
      Sub(in1 := #"RECETA  EQUIPOS"[#"NUMERO EQUIPO"]."TEMP AGUA"[#"PASO ACTUAL"[#"NUMERO EQUIPO"]], in2 := #CONFIGURACIONES[#"NUMERO EQUIPO"].HISTERESIS, out => #"HISTERESIS MINIMA"[#"NUMERO EQUIPO"])
   END_RUNG
   RUNG wire#powerrail
      Move(in := #"HISTERESIS MINIMA"[#"NUMERO EQUIPO"], out1 => #"SALIDA HISTERESIS MINIMA"[#"NUMERO EQUIPO"])
   END_RUNG
   RUNG wire#powerrail
      Contact( #"INICIAR CICLO OP"[#"NUMERO EQUIPO"] )
      Contact( #"TIPO DE EQUIPO"[#"NUMERO EQUIPO"] )
      { S7_Templates := "SrcType := Real" } LT_Contact(in1 := #TEMPERATURAS[#"NUMERO EQUIPO"]."TEMPERATURA AGUA", in2 := #"HISTERESIS MINIMA"[#"NUMERO EQUIPO"])
      S_SR(operand := #"AUXILIAR VS"[#"NUMERO EQUIPO"], r1 := wire#w1)
   END_RUNG
   RUNG wire#powerrail
      Contact( #"INICIAR CICLO OP"[#"NUMERO EQUIPO"] )
      Contact( #"TIPO DE EQUIPO"[#"NUMERO EQUIPO"] )
      { S7_Templates := "SrcType := Real" } GT_Contact(in1 := #TEMPERATURAS[#"NUMERO EQUIPO"]."TEMPERATURA AGUA", in2 := #"HISTERESIS MAXIMA"[#"NUMERO EQUIPO"])
   END_RUNG wire#w1
   RUNG wire#powerrail
      Contact( #"PAUSAR CICLO"[#"NUMERO EQUIPO"] )
   END_RUNG wire#w1
   RUNG wire#powerrail
      Contact( #"CICLO CANCELADO"[#"NUMERO EQUIPO"] )
   END_RUNG wire#w1
   // the same network as SCL:
   #"HISTERESIS MAXIMA"[#"NUMERO EQUIPO"] := #"RECETA  EQUIPOS"[#"NUMERO EQUIPO"]."TEMP AGUA"[#"PASO ACTUAL"[#"NUMERO EQUIPO"]] + #CONFIGURACIONES[#"NUMERO EQUIPO"].HISTERESIS;
   #"SALIDA HISTERESIS MAXIMA"[#"NUMERO EQUIPO"] := #"HISTERESIS MAXIMA"[#"NUMERO EQUIPO"];
   #"HISTERESIS MINIMA"[#"NUMERO EQUIPO"] := #"RECETA  EQUIPOS"[#"NUMERO EQUIPO"]."TEMP AGUA"[#"PASO ACTUAL"[#"NUMERO EQUIPO"]] - #CONFIGURACIONES[#"NUMERO EQUIPO"].HISTERESIS;
   #"SALIDA HISTERESIS MINIMA"[#"NUMERO EQUIPO"] := #"HISTERESIS MINIMA"[#"NUMERO EQUIPO"];
   #_w1 := (#"INICIAR CICLO OP"[#"NUMERO EQUIPO"] AND #"TIPO DE EQUIPO"[#"NUMERO EQUIPO"] AND (#TEMPERATURAS[#"NUMERO EQUIPO"]."TEMPERATURA AGUA" > #"HISTERESIS MAXIMA"[#"NUMERO EQUIPO"])) OR #"PAUSAR CICLO"[#"NUMERO EQUIPO"] OR #"CICLO CANCELADO"[#"NUMERO EQUIPO"];
   IF #"INICIAR CICLO OP"[#"NUMERO EQUIPO"] AND #"TIPO DE EQUIPO"[#"NUMERO EQUIPO"] AND (#TEMPERATURAS[#"NUMERO EQUIPO"]."TEMPERATURA AGUA" < #"HISTERESIS MINIMA"[#"NUMERO EQUIPO"]) THEN
       #"AUXILIAR VS"[#"NUMERO EQUIPO"] := TRUE;   // SR flip-flop
   END_IF;
   IF #_w1 THEN #"AUXILIAR VS"[#"NUMERO EQUIPO"] := FALSE; END_IF;
END_REGION

